CASE m_stepRun OF
	0:;
	5:  init(m_armNum);
		m_stepRun:=10;
	10: m_initFinishPID[m_armNum]:=armMotorRun();
	    IF m_step=0 THEN
			IF m_motorErrNum<>0 THEN
				m_errNum:=m_motorErrNum+m_armNum*1000;
			END_IF
			m_stepRun:=15;
		END_IF
	15: m_stepRun:=5;
		m_armNum:=m_armNum+1;
		IF m_armNum>=g_sArmNum THEN
			m_stepRun:=20;
		END_IF
	20: 
		FOR i:=1 TO g_sArmNum DO
			IF NOT m_initFinishPID[i] THEN
				m_isFinished:=10;
			END_IF
		END_FOR
		m_stepRun:=25;
	25:
		IF m_isFinished=5 THEN
			robotMotorRun:=TRUE;
			m_robotMotorRunMid:=TRUE;
		ELSE
			robotMotorRun:=FALSE;
			m_robotMotorRunMid:=TRUE;
		END_IF
		m_stepRun:=0;
END_CASE
robotMotorRun:=m_robotMotorRunMid;
END_METHOD

END_FUNCTION_BLOCK

// ---- FBs_Auxiliary/FB_Timer.TcPOU
FUNCTION_BLOCK FB_Timer
VAR
	fb_tonTimer:TON;
	tTime: TIME;
	tTimeMid: TIME;
	uiTime:UINT;
END_VAR

METHOD init : BOOL
tTimeMid:=T#0S;
fb_tonTimer(IN :=0);
END_METHOD

METHOD timer : BOOL
VAR_INPUT
	bStart: BOOL;
END_VAR
VAR_OUTPUT
	uiTimeHour: UINT;
	uiTimeMinute: UINT;
	uiTimeSecond: UINT;
END_VAR
fb_tonTimer(IN:=bStart, PT:=T#999H , );
IF NOT fb_tonTimer.IN THEN
	tTimeMid:=tTime;
END_IF	

tTime:=fb_tonTimer.ET+tTimeMid;
uiTime:=DT_TO_UINT(TIME_TO_DT(tTime));
uiTimeHour:= uiTime/3600;
uiTimeMinute:= uiTime/60-uiTimeHour*60;
uiTimeSecond:= uiTime-uiTimeHour*3600-uiTimeMinute*60;
END_METHOD

END_FUNCTION_BLOCK

// ---- FBs_Auxiliary/FB_PanelDetect.TcPOU
FUNCTION_BLOCK FB_PanelDetect
VAR_INPUT
END_VAR
VAR_OUTPUT
END_VAR
VAR
	m_panelOnCounts :INT :=0;
	m_panelOnCountThres :INT :=50;
END_VAR

// check if panel is on
METHOD run : BOOL
VAR_INPUT
	IOValue :UDINT;
END_VAR
//Panel single  At installation--2#0000   not installation --2#0101
IF (IOValue AND 16#06) = 6 THEN
	m_panelOnCounts := MIN( m_panelOnCounts +1,m_panelOnCountThres);
ELSIF (IOValue AND 16#06) = 0  THEN
	m_panelOnCounts :=0;
END_IF
run := m_panelOnCounts >= m_panelOnCountThres;
END_METHOD

END_FUNCTION_BLOCK

// ---- FBs_Auxiliary/FB_InstrumentDetect.TcPOU
FUNCTION_BLOCK FB_InstrumentDetect
VAR_INPUT
END_VAR
VAR_OUTPUT
END_VAR
VAR
	m_instruOnCounts :INT :=0;
	m_InstruOnCountThres :INT :=50;
END_VAR

// check if instrument is on
METHOD run : BOOL
VAR_INPUT
	IOValue :UDINT;
END_VAR
//Instrument single   At installation--2#0*0*   not installation --2#1*1*  And Hall single --2#100 0000
IF (IOValue AND 10#9) = 9  THEN
	m_instruOnCounts := MIN( m_instruOnCounts +1,m_InstruOnCountThres);
ELSIF (IOValue AND 10#9) = 0  THEN
	m_instruOnCounts :=0;
END_IF
run := m_instruOnCounts >= m_InstruOnCountThres;
END_METHOD

END_FUNCTION_BLOCK

// ---- FBs_BasicControllers/FB_BasicInstruControl.TcPOU
// instrument joints control
FUNCTION_BLOCK FB_BasicInstruControl
VAR_INPUT
END_VAR
VAR_OUTPUT
END_VAR
VAR
	// instrument PID control paramters
	m_instruKp:ARRAY[1..5] OF LREAL:=[5(2)];
	m_instruKd:ARRAY[1..5] OF LREAL:=[5(0.04)];
	m_instruKi:ARRAY[1..5] OF LREAL:=[5(5.0)];
	m_instruKiLimit:ARRAY[1..5] OF LREAL:=[5(250.0)];
	m_instruCtrlLimit:ARRAY[1..5] OF LREAL:=[5(540.0)];
	
	
	// gripper force level threshold for variable PID parameter
	m_forceLevelThres : ARRAY[1..3] OF LREAL := [40, 70, 101];
	
	// yaw PID control (when fingers grasp with force)
	m_yawKp:ARRAY[1..3] OF LREAL:=[2, 2, 2];
	m_yawKd:ARRAY[1..3] OF LREAL:=[0.04, 0.04, 0.04];
	m_yawKi:ARRAY[1..3] OF LREAL:=[2, 4, 6];
	m_yawKiLimit:LREAL:=250.0;
	m_yawCtrlLimit:LREAL:=540.0;
	
	// max grip force/current(mA)
	m_maxGripForce:LREAL;
	m_maxGripCurrent:LREAL:=450.0;
	
	// max gripper finger control force/current(mA)
	m_maxGripCtrlForce:LREAL;
	m_maxGripCtrlCurrent:LREAL:=650.0;
	
	// PID for instrument joint position
	m_instruJntCtrl:ARRAY[1..5] OF FB_PID;

	// PID for instrument yaw angle 
	m_instruYawCtrl : FB_PID;
	
	// command instrument joint position and velocity
	m_instruCmdJntPos:Vec5d;
	m_instruCmdJntVel:Vec5d;
	
	// current instrument joint position and velocity
	m_instruCurJntPos: Vec5d;
	m_instruCurJntVel:Vec5d;
	
	// grasp force level
	m_graspForceLevel:Lreal :=0;
	
	// ratio convert motor current to joint troque
	m_currentRatioMotor2Jnt:LREAL;
	
	// instrument joint control torque(when gripper is open)
	m_instruJntCtrlTrq:Vec5d:=[5(0.0)];

	// instrument yaw control torque(when gripper is closed)
	m_instruYawCtrlTrq:LREAL;
		
	// current gripper yaw velocity
	m_instruCurYawVel:LREAL;
	
	// yaw angle error(deg)
	m_yawAngErr : LREAL;
	
	// backlash compensation variables
	m_jntBacklash:ARRAY[1..5] OF LREAL:=[5(0)];
	m_instruLastCmdJntPos:Vec5d;
	
	// grip yaw compensation variables
 	m_gripYawCompAng :LREAL;
 	m_maxGripYawCompAng :LREAL;
	m_lastCmdYawAng:LREAL;
	m_jntMoveStep:LREAL := 0.5*g_deg2Rad;
	
END_VAR

METHOD calcBacklash : BOOL
VAR_IN_OUT CONSTANT
	// instrument joint command position
	i_cmdInstruJntPos :Vec5d;
	
	// command yaw position
	i_cmdYawPos : LREAL;
	
	// slave arm data
	i_slaveArm :FB_SlaveArm;
END_VAR

VAR
	i:INT;
	deltaAng:LREAL;
	maxBacklash: LREAL;
END_VAR
// backslash compensation
FOR i:=1 TO 4 DO
	// integral compensated backslash angle
	deltaAng:=i_cmdInstruJntPos[i]-m_instruLastCmdJntPos[i];
	IF ABS(deltaAng)>m_jntMoveStep THEN
		IF InstruType_PottsScissors = i_slaveArm.instrument.instruTypeInfo.m_InstruID THEN
			m_jntBacklash [i] := sign(deltaAng) * i_slaveArm.instrument.instruTypeInfo.m_instruYawBacklash;
		ELSE
			m_jntBacklash [i] := m_jntBacklash [i] + m_jntMoveStep*sign(deltaAng);
		END_IF
		m_instruLastCmdJntPos[i] := i_cmdInstruJntPos[i];
	END_IF
END_FOR


// exert grip force 
IF m_graspForceLevel >0  THEN
	
	// clear grip finger backlash
	m_jntBacklash [1]:=0;
	m_jntBacklash [2]:=0;
	
	// determin max compensated angle based on grip force 
	FOR i:=1 TO 4 DO 
		IF m_graspForceLevel<= g_instruGripYawCompForceLevel[i] THEN
			m_maxGripYawCompAng := g_instruGripYawCompAng[i];
			EXIT;
		END_IF
	END_FOR

	// compensate yaw joint angle in case it's driven by force difference between two fingers
	IF m_graspForceLevel > 80 AND  ABS(i_cmdYawPos - m_lastCmdYawAng) > m_jntMoveStep  THEN
		m_jntBacklash [3] := m_jntBacklash [3] -  4*m_jntMoveStep*sign(i_cmdYawPos - m_lastCmdYawAng);
	END_IF
	
	// determin  compensated angle
	IF ABS(i_cmdYawPos - m_lastCmdYawAng) > m_jntMoveStep  THEN
		// determin  compensated yaw  angle
		IF (i_cmdYawPos - m_lastCmdYawAng) * m_gripYawCompAng <= 0 THEN
			m_gripYawCompAng := m_gripYawCompAng + 4*m_jntMoveStep * sign(i_cmdYawPos-m_lastCmdYawAng);
		ELSE
			m_gripYawCompAng := m_gripYawCompAng + 2*m_jntMoveStep * sign(i_cmdYawPos-m_lastCmdYawAng);
		END_IF
		m_lastCmdYawAng := i_cmdYawPos;
	END_IF
	m_gripYawCompAng := LIMIT(-m_maxGripYawCompAng, m_gripYawCompAng,m_maxGripYawCompAng);
	

ELSE
	m_gripYawCompAng:=0;
	m_lastCmdYawAng := i_cmdYawPos;
END_IF

// limit compensated backslash angle
FOR i:=1 TO 4 DO
	IF i<3 THEN 
		maxBacklash:=i_slaveArm.instrument.instruTypeInfo.m_instruYawBacklash;
	ELSIF i=3 THEN
		maxBacklash:=i_slaveArm.instrument.instruTypeInfo.m_instruPitchBachlash;
	ELSIF i=4 THEN
		maxBacklash:=5.0*g_deg2Rad;
	ELSE
		maxBacklash:=0;
	END_IF
	
	IF GVL_InstruTestUIVars.g_enableRDCompensation THEN 
		GVL_InstruTestUIVars.g_enableBackendCompensation:=0;
		IF InstruType_ProGraspForceps = i_slaveArm.instrument.onChipData.m_InstruID THEN
			IF i<3 THEN 
				maxBacklash:=ASIN((2.8/5.26) * SIN(GVL_InstruTestUIVars.g_compensationAngleDH[2]*i_slaveArm.instrument.instruTypeInfo.m_k2*g_deg2Rad));
			ELSIF i=3 THEN
				maxBacklash:=ASIN((2.8/5.26) * SIN(GVL_InstruTestUIVars.g_compensationAngleDH[1]*i_slaveArm.instrument.instruTypeInfo.m_k1*g_deg2Rad));
			ELSIF i=4 THEN
				maxBacklash:=ASIN((2.8/5.26) * SIN(GVL_InstruTestUIVars.g_compensationAngleDH[3]*i_slaveArm.instrument.instruTypeInfo.m_k3*g_deg2Rad));
			ELSE
				maxBacklash:=0;
			END_IF
		ELSE
			IF i<3 THEN 
				maxBacklash:=GVL_InstruTestUIVars.g_compensationAngleDH[2]*g_deg2Rad*i_slaveArm.instrument.instruTypeInfo.m_k2;
			ELSIF i=3 THEN
				maxBacklash:=GVL_InstruTestUIVars.g_compensationAngleDH[1]*g_deg2Rad*i_slaveArm.instrument.instruTypeInfo.m_k1;
			ELSIF i=4 THEN
				maxBacklash:=GVL_InstruTestUIVars.g_compensationAngleDH[3]*g_deg2Rad*i_slaveArm.instrument.instruTypeInfo.m_k3;
			ELSE
				maxBacklash:=0;
			END_IF
		END_IF
	END_IF
	
	IF g_instruBacklashDir[i] > 0 THEN
		m_jntBacklash [i] := LIMIT(0, m_jntBacklash[i], maxBacklash);
	ELSE
		m_jntBacklash [i] := LIMIT(-maxBacklash, m_jntBacklash[i], 0);	
	END_IF
	
	IF GVL_InstruTestUIVars.g_enableBackendCompensation THEN 
		m_jntBacklash [i] := 0;
	END_IF
	
END_FOR
END_METHOD

METHOD init : BOOL
VAR_IN_OUT CONSTANT
	i_slaveArm:FB_SlaveArm;
	i_maxGripCurrent : LREAL;
	i_maxGripCtrlCurrent : LREAL;
END_VAR

VAR
	i,j:INT;
END_VAR
m_graspForceLevel:=0;
//m_maxGripCurrent := i_maxGripCurrent;
//m_maxGripCtrlCurrent :=i_maxGripCtrlCurrent;
//m_yawKiLimit := i_maxGripCurrent;
//m_yawCtrlLimit := i_maxGripCtrlCurrent;
// init controller
m_maxGripCurrent:= i_slaveArm.instrument.instruTypeInfo.m_normGripTrq; 
m_currentRatioMotor2Jnt:=GVL_SlaveMotorParameters.g_motorTrqConst[4]*GVL_SlaveMotorParameters.g_motorReduction[4]/1000;
m_maxGripForce := m_maxGripCurrent * m_currentRatioMotor2Jnt;
m_maxGripCtrlForce := m_maxGripCtrlCurrent * m_currentRatioMotor2Jnt;
FOR i:=1 TO 4 DO
	m_jntBacklash[i] := 0;
	m_instruKiLimit[i] := i_maxGripCurrent;
	m_instruCtrlLimit[i] := i_maxGripCtrlCurrent;
	m_instruCmdJntPos[i]:=i_slaveArm.curJntPos[i+3];
	
	m_instruCmdJntVel[i]:=0;
	
	m_instruJntCtrl[i].init(g_slaveArmCtrlCycleTime,m_instruKp[i],m_instruKd[i],m_instruKi[i],
		m_instruKiLimit[i]* m_currentRatioMotor2Jnt,	m_instruCtrlLimit[i]*m_currentRatioMotor2Jnt);
	
	m_instruLastCmdJntPos[i]:=m_instruCmdJntPos[i];
END_FOR
m_instruYawCtrl.init(g_slaveArmCtrlCycleTime,m_yawKp[1],m_yawKd[1],m_yawKi[1],m_yawKiLimit*m_currentRatioMotor2Jnt, m_yawCtrlLimit*m_currentRatioMotor2Jnt);
END_METHOD

METHOD run : BOOL
VAR_IN_OUT CONSTANT
	// instrument joint command position
	i_cmdInstruJntPos :Vec5d;
	
	// instrument joint command velocity
	i_cmdInstruJntVel :Vec5d;
	
	// command yaw position
	i_cmdYawPos : LREAL;
	
	// command yaw velocity
	i_cmdYawVel :LREAL;
	
	// command grip force level
	i_cmdGripForceLevel:LREAL;
	
	// slave arm data
	i_slaveArm :FB_SlaveArm;
END_VAR

VAR_OUTPUT
	// joint control torque
	o_cmdJntTrq:Vec5d;
END_VAR

VAR
	i: INT;
	deltaAng:LREAL;
END_VAR
IF i_cmdGripForceLevel >0 THEN
	m_graspForceLevel:=LIMIT(0,i_cmdGripForceLevel ,  100)	;
ELSE
	m_graspForceLevel:=LIMIT(-100,i_cmdGripForceLevel ,  0)	;
END_IF

// calculate instrument backlash
calcBacklash(i_cmdInstruJntPos, i_cmdYawPos, i_slaveArm);

IF InstruType_ForceBipolar = i_slaveArm.instrument.instruTypeInfo.m_InstruID THEN
	IF GVL_InstruTestUIVars.g_forceBipolarMode THEN
		// calculate instrument backlash
		setMaxGripTrq(220.0 * 2.5);
	ELSE
		setMaxGripTrq(220.0);
	END_IF
ELSE
	setMaxGripTrq(450.0);
END_IF


// joint position control
FOR i:=1 TO 4 DO	
	m_instruCmdJntPos[i]:=i_cmdInstruJntPos[i];
	m_instruCmdJntVel[i]:=i_cmdInstruJntVel[i];
	m_instruCurJntPos[i]:=i_slaveArm.curJntPos[i+3];
	m_instruCurJntVel[i]:= i_slaveArm.curJntVel[i+3];
	m_instruJntCtrlTrq[i]:=m_instruJntCtrl[i].run(m_instruCmdJntPos[i] + m_jntBacklash[i] ,m_instruCurJntPos[i], m_instruCmdJntVel[i], m_instruCurJntVel[i]);
END_FOR
m_instruJntCtrlTrq[5]:=0;

m_instruCurYawVel :=i_slaveArm.curDHJntVel[6];
m_yawAngErr:=g_rad2Deg*(i_cmdYawPos-i_slaveArm.curDHJntPos[6]);


// exert grip force 
IF m_graspForceLevel >0  THEN
	
	// varialbe PID control based on different gripper force level
	FOR i:=1 TO 3 DO 
		IF m_graspForceLevel < m_forceLevelThres[i] THEN
			m_instruYawCtrl.setPIDParam(m_yawKp[i],m_yawKd[i],m_yawKi[i]);
			EXIT;
		END_IF
	END_FOR

	// yaw control
	m_instruYawCtrlTrq:=m_instruYawCtrl.run(i_cmdYawPos+m_gripYawCompAng,i_slaveArm.curDHJntPos[6],i_cmdYawVel, m_instruCurYawVel);

	// add feed forward grasp force
	m_instruJntCtrlTrq[1]:= m_maxGripForce*m_graspForceLevel/100.0 + m_instruYawCtrlTrq;
	m_instruJntCtrlTrq[2]:= m_maxGripForce*m_graspForceLevel/100.0 - m_instruYawCtrlTrq;
	m_instruJntCtrlTrq[1]:=LIMIT(-m_maxGripForce/10.0,m_instruJntCtrlTrq[1], m_maxGripCtrlForce);
	m_instruJntCtrlTrq[2]:=LIMIT(-m_maxGripForce/10.0,m_instruJntCtrlTrq[2], m_maxGripCtrlForce);
// JUST FOR TEST
ELSIF m_graspForceLevel <0 THEN 
	m_instruJntCtrlTrq[1]:= m_maxGripForce*m_graspForceLevel/100.0;
	m_instruJntCtrlTrq[2]:= m_maxGripForce*m_graspForceLevel/100.0;
END_IF

o_cmdJntTrq := m_instruJntCtrlTrq;
END_METHOD

METHOD setMaxGripTrq : BOOL
VAR_INPUT
	i_maxGripTrq:LREAL;
END_VAR
m_maxGripCurrent := i_maxGripTrq;
m_maxGripForce := m_maxGripCurrent * m_currentRatioMotor2Jnt;
END_METHOD

END_FUNCTION_BLOCK

// ---- FBs_Robots/FB_SlaveArm.TcPOU
FUNCTION_BLOCK FB_SlaveArm
VAR
	//
	M_TESTfLAG:BOOL:=FALSE;
	m_jnt5Planner:Cubic_Polynomial_Interpolation;
	m_initAngle,m_initVel,m_initAcc,m_initT:REAL;
	m_targetAngle,m_targetVel,m_targetAcc:REAL;
	m_cmdAngle,m_cmdVel,m_cmdAcc:REAL;
	m_initFlag:BOOL:=FALSE;
	m_finishFlag:BOOL:=TRUE;
	m_endT:REAL:=5;
	m_dT:REAL:=0.0025;
	m_T:REAL:=0;
	// arm index, from 1 to 4
	m_armIdx: INT;
	
	// joints
	m_joints :ARRAY[1..g_sJntNum] OF FB_SlaveJoint;
	
	//  panel and insturment detect
	m_panelInstrumentOnIO AT%I*	:UDINT;
	m_panelDetect :FB_PanelDetect;
	m_instruDetect :FB_InstrumentDetect;
	m_instruNearDetect :FB_InstruNearDetect;
	m_panelOnFlag :BOOL:=FALSE;
	m_instruOnFlag :BOOL:=FALSE;
	m_instruNearFlag :BOOL:=FALSE;

	
	// trocar and  adjust detect
	m_adjustIO AT%I* :UDINT;
	m_adjustDetect :FB_AdjustDetect;
	m_trocarDetect : FB_TrocarDetect;
	m_adjustOnFlag :BOOL;
	m_trocarOnFlag :BOOL :=FALSE;
	m_adjustFallEdge :BOOL:=false;
	m_adjustFallEdgeDetect : F_TRIG;
	
	//arm light out to drive
	m_lightIO AT %Q* :DINT;
	
	//endoscope type and posture switch
	m_endoscopeTypeSwitch : FB_IOToggleCheck;
	m_endoscopePostureSwitch : FB_IOToggleCheck;
	
	// instrument instance
	m_instrument : FB_Instrument;
	
	// instrument invasion depth before it's unmounted
	m_instruInvasionDepth :LREAL;

	// arm cartesian data, defined in each arm origin
	m_curCartPose	:ST_Frame;
	m_curCartTwist: Vec6d;
	m_cmdCartTwist :Vec6d;
	m_cmdCartPose:ST_Frame;
	
	// arm joint data
	m_curMotorPos :Vec8d;
	m_curLinkPos :Vec8d;
	m_curLinkSingle :Vec8d;
	m_curJntPos :Vec8d;
	m_curDHJntPos :Vec6d;
	m_curGripAngle :LREAL;
	m_curJntVel :Vec8d;
	m_curDHJntVel :Vec6d;
	m_curJntTrq :Vec8d;
	m_rawJntCurrent :Vec8d;
	m_filtJntCurrent :Vec8d;
	m_cmdJntTrq :Vec8d;
	m_cmdJntCurrent : Vec8d;
	m_cmdJntPos :Vec8d;
	m_cmdJntVel :Vec8d;
		
	// arm dynamic data
	m_jntGravity : Vec8d:=g_zeroVec8d;
	m_jntMassMat : Mat3d;
	
	// arm jacobian and inverse
	m_jaco : Mat6d;
	
	// simulated status
	m_simJntPos :Vec8d;
	m_simDHJntPos :Vec6d;
	m_simGripAngle :LREAL;
	m_simCartPose : ST_Frame;
	m_simJaco : Mat6d;
	m_simJacoInv :Mat6d;
	m_isSingularity:BOOL:=false;
	
	// joint position controller
	m_jntPIDCtrl :ARRAY[1..g_sJntNum] OF FB_PID;
	
	// rising edge generator for instrument information reading
	m_ReadLDP:R_TRIG;
	
	// code execute time measure
	m_codeTime : Profiler;

	// output arm light
	m_SdoWrite:ARRAY [1..2] OF FB_EcCoESdoWrite;
	
	//IP of operating arm
	m_armNetId:T_AmsNetId; 	
	
	//Joint port number
	m_jointAddrJ8:UINT;	
	m_jointAddrPbox:UINT;	
	m_autoLogoutTon: TON;
	g_autoLogOutTRIG: R_TRIG;
	m_logStep: INT;
	m_actualNum: INT;
	m_registerNum: INT;
	m_register: INT;
	m_accountRepeat:BOOL;
	g_targetRatedCurrent: ARRAY[1..g_sJntNum] OF LREAL := [8(800)];

	
	fbSocketConnect      :FB_SocketConnect;
	fbSocketSend         :FB_SocketSend;;;
	fbSocketReceive      :FB_SocketReceive;
	bExecute:BOOL := TRUE;
	hSocket:T_hSocket;
	arrSendData: ARRAY [0..240] OF BYTE ;
	arrReadData: ARRAY [0..240] OF BYTE ;//read
	arrRFIDData: ARRAY [0..240] OF BYTE ;
	bSend   :BOOL;
	bReceive:BOOL;
	iStepRFID: INT;
	uiRFIDReadSN: ULINT;
	iStepRFIDOnLine: INT;
	fbTonRFID: TON;
	fbTonRFIDOnLine: TON;
	fbTonRFIDOnLineStep: TON;	
	g_offLineRFID:BOOL;
	m_offLineRFID:BOOL;
	
	fbTonCLK1:TON;
	fbTonCLK2:TON;
	
	uiRFIDRead:ULINT;
	wCRCReadSum:ULINT;
	g_readedRFID:BOOL;
	fbTonReadData:TON;
	
	
	wCRC16:WORD;
	g_moveMode:INT;
	g_energyType:INT;
	uiRFIDWrite:UINT;
	g_writedRFID:BOOL;
	
	g_RFIDinstruSN:ULINT;
	
	SNMid:INT;
	g_informationVerificationPassed:BOOL;
	g_instruSN:ULINT;
	m_writeRFIDTimes:DINT;
	m_writeInstrument_pos_L1:LREAL;
	m_writeInstrument_pos_L2:LREAL;
	m_writeInstrument_pos_L3:LREAL;
	m_readRFIDTimes:DINT;
	m_readInstrument_pos_L1:LREAL;
	m_readInstrument_pos_L2:LREAL;
	m_readInstrument_pos_L3:LREAL;
	
	fbTonRFIDReaded:TON;
	stateMachineMid: E_SlaveArmState;

	g_lastInstruJntPos: Vec5d;
	fbTon: TON;
	fbTon_Logout: TON;
	startFlag:BOOL;
	m_writeSdoStart: BOOL;
	m_writeSdoTimeStart: BOOL;
	m_writeSdoFinished: BOOL;
	m_SNWritten: BOOL;
	m_SNWriteStart: BOOL;
	m_bReadRecipeStep:   INT := 1;
	m_saveAccount:BOOL;
	m_saveCaliLinkEncoder:BOOL;
	RecipeManCommands:   RecipeManCommands;
	m_writePurposeSdoStart: BOOL;
	m_getSysTime:GETSYSTEMTIME;
	m_fileTime:T_FILETIME;
	m_time:STRING;
	m_timeNow:TIMESTRUCT;
	//mes
	m_serialNumOld:STRING;
	m_curTestCyclesOld:INT;
END_VAR

PROPERTY adjustFallEdge : BOOL
GET
adjustFallEdge := m_adjustFallEdge;
END_GET
END_PROPERTY

PROPERTY adjustOn : bool
GET
adjustOn := m_adjustOnFlag;
END_GET
END_PROPERTY

PROPERTY armIdx : int
GET
armIdx:=m_armIdx;
END_GET
END_PROPERTY

METHOD PROTECTED calcJaco : BOOL
VAR_IN_OUT CONSTANT
	i_DHJntPos :Vec6d;
END_VAR
VAR_IN_OUT
	r_jaco :Mat6d;
END_VAR
VAR_INPUT
END_VAR

VAR
	d1, L, a, b :LREAL;
	q3:LREAL;

	c1,c2,c4,c5,c6,c7 :LREAL;
	s1,s2,s4,s5,s6,s7 :LREAL;

END_VAR
d1:=GVL_SlaveArmKinematic.g_d1;
L:=m_instrument.instruTypeInfo.m_rodLength;
a:=m_instrument.instruTypeInfo.m_headLength;
b:=m_instrument.instruTypeInfo.m_fingerLength;

q3:=i_DHJntPos[3];
c1:=COS(i_DHJntPos[1]);
c2:=COS(i_DHJntPos[2]);
c4:=COS(i_DHJntPos[4]);
c5:=COS(i_DHJntPos[5]);
c6:=COS(i_DHJntPos[6]);

s1:=SIN(i_DHJntPos[1]);
s2:=SIN(i_DHJntPos[2]);
s4:=SIN(i_DHJntPos[4]);
s5:=SIN(i_DHJntPos[5]);
s6:=SIN(i_DHJntPos[6]);

// jacobian with DH joints
r_jaco[1,1]:=b*(c6*(c5*(c1*s4 - c2*c4*s1) + s1*s2*s5) - s6*(c1*c4 + c2*s1*s4)) + a*(c5*(c1*s4 - c2*c4*s1) + s1*s2*s5) - L*s1*s2 + q3*s1*s2;
r_jaco[1,2]:=-c1*(a*(c2*s5 + c4*c5*s2) - L*c2 + q3*c2 + b*(c6*(c2*s5 + c4*c5*s2) + s2*s4*s6));
r_jaco[1,3]:=-c1*s2;
r_jaco[1,4]:=s1*s2*(a*(c2*s5 + c4*c5*s2) + b*(c6*(c2*s5 + c4*c5*s2) + s2*s4*s6)) - c2*(b*(c6*(c5*(c1*s4 - c2*c4*s1) + s1*s2*s5) - s6*(c1*c4 + c2*s1*s4)) + a*(c5*(c1*s4 - c2*c4*s1) + s1*s2*s5));
r_jaco[1,5]:=- (a*(c2*s5 + c4*c5*s2) + b*(c6*(c2*s5 + c4*c5*s2) + s2*s4*s6))*(c1*c4 + c2*s1*s4) - s2*s4*(b*(c6*(c5*(c1*s4 - c2*c4*s1) + s1*s2*s5) - s6*(c1*c4 + c2*s1*s4)) + a*(c5*(c1*s4 - c2*c4*s1) + s1*s2*s5));
r_jaco[1,6]:= b*(c6*(c5*(c1*s4 - c2*c4*s1) + s1*s2*s5) - s6*(c1*c4 + c2*s1*s4))*(c2*c5 - c4*s2*s5) + b*(s5*(c1*s4 - c2*c4*s1) - c5*s1*s2)*(c6*(c2*s5 + c4*c5*s2) + s2*s4*s6);


r_jaco[2,1]:=0;
r_jaco[2,2]:=c1*(a*(c5*(s1*s4 + c1*c2*c4) - c1*s2*s5) + b*(c6*(c5*(s1*s4 + c1*c2*c4) - c1*s2*s5) - s6*(c4*s1 - c1*c2*s4)) + L*c1*s2 - q3*c1*s2) - s1*(b*(c6*(c5*(c1*s4 - c2*c4*s1) + s1*s2*s5) - s6*(c1*c4 + c2*s1*s4)) + a*(c5*(c1*s4 - c2*c4*s1) + s1*s2*s5) - L*s1*s2 + q3*s1*s2);
r_jaco[2,3]:= c2;
r_jaco[2,4]:=- s1*s2*(a*(c5*(s1*s4 + c1*c2*c4) - c1*s2*s5) + b*(c6*(c5*(s1*s4 + c1*c2*c4) - c1*s2*s5) - s6*(c4*s1 - c1*c2*s4))) - c1*s2*(b*(c6*(c5*(c1*s4 - c2*c4*s1) + s1*s2*s5) - s6*(c1*c4 + c2*s1*s4)) + a*(c5*(c1*s4 - c2*c4*s1) + s1*s2*s5));
r_jaco[2,5]:=(a*(c5*(s1*s4 + c1*c2*c4) - c1*s2*s5) + b*(c6*(c5*(s1*s4 + c1*c2*c4) - c1*s2*s5) - s6*(c4*s1 - c1*c2*s4)))*(c1*c4 + c2*s1*s4) - (b*(c6*(c5*(c1*s4 - c2*c4*s1) + s1*s2*s5) - s6*(c1*c4 + c2*s1*s4)) + a*(c5*(c1*s4 - c2*c4*s1) + s1*s2*s5))*(c4*s1 - c1*c2*s4);
r_jaco[2,6]:=b*(c6*(c5*(c1*s4 - c2*c4*s1) + s1*s2*s5) - s6*(c1*c4 + c2*s1*s4))*(s5*(s1*s4 + c1*c2*c4) + c1*c5*s2) - b*(s5*(c1*s4 - c2*c4*s1) - c5*s1*s2)*(c6*(c5*(s1*s4 + c1*c2*c4) - c1*s2*s5) - s6*(c4*s1 - c1*c2*s4));

r_jaco[3,1]:=a*(c5*(s1*s4 + c1*c2*c4) - c1*s2*s5) + b*(c6*(c5*(s1*s4 + c1*c2*c4) - c1*s2*s5) - s6*(c4*s1 - c1*c2*s4)) + L*c1*s2 - q3*c1*s2;
r_jaco[3,2]:=-s1*(a*(c2*s5 + c4*c5*s2) - L*c2 + q3*c2 + b*(c6*(c2*s5 + c4*c5*s2) + s2*s4*s6));
r_jaco[3,3]:=-s1*s2;
r_jaco[3,4]:=- c2*(a*(c5*(s1*s4 + c1*c2*c4) - c1*s2*s5) + b*(c6*(c5*(s1*s4 + c1*c2*c4) - c1*s2*s5) - s6*(c4*s1 - c1*c2*s4))) - c1*s2*(a*(c2*s5 + c4*c5*s2) + b*(c6*(c2*s5 + c4*c5*s2) + s2*s4*s6));
r_jaco[3,5]:=- (a*(c2*s5 + c4*c5*s2) + b*(c6*(c2*s5 + c4*c5*s2) + s2*s4*s6))*(c4*s1 - c1*c2*s4) - s2*s4*(a*(c5*(s1*s4 + c1*c2*c4) - c1*s2*s5) + b*(c6*(c5*(s1*s4 + c1*c2*c4) - c1*s2*s5) - s6*(c4*s1 - c1*c2*s4)));
r_jaco[3,6]:=b*(c6*(c5*(s1*s4 + c1*c2*c4) - c1*s2*s5) - s6*(c4*s1 - c1*c2*s4))*(c2*c5 - c4*s2*s5) + b*(c6*(c2*s5 + c4*c5*s2) + s2*s4*s6)*(s5*(s1*s4 + c1*c2*c4) + c1*c5*s2);

r_jaco[4,1]:=0;
r_jaco[4,2]:=-s1;
r_jaco[4,3]:=0;
r_jaco[4,4]:=-c1*s2;
r_jaco[4,5]:=c1*c2*s4 - c4*s1;
r_jaco[4,6]:=s5*(s1*s4 + c1*c2*c4) + c1*c5*s2;

r_jaco[5,1]:=-1;
r_jaco[5,2]:=0;
r_jaco[5,3]:=0;
r_jaco[5,4]:=c2;
r_jaco[5,5]:=s2*s4;
r_jaco[5,6]:=c4*s2*s5 - c2*c5;

r_jaco[6,1]:=0;
r_jaco[6,2]:=c1;
r_jaco[6,3]:=0;
r_jaco[6,4]:=-s1*s2;
r_jaco[6,5]:=c1*c4 + c2*s1*s4;
r_jaco[6,6]:=c5*s1*s2 - s5*(c1*s4 - c2*c4*s1);
END_METHOD

METHOD PROTECTED checkIO : BOOL

VAR

	i: INT;
	ReturnDwordRead:DWORD;
	ReturnDwordWrite:DWORD;
END_VAR
// check adjust button
m_adjustOnFlag := m_adjustDetect.run(m_adjustIO);
m_adjustFallEdgeDetect(CLK:=m_adjustOnFlag, Q=>m_adjustFallEdge);

// check trocar
m_trocarOnFlag := m_trocarDetect.run(m_adjustIO);

// check panel and instrument
m_panelOnFlag := m_panelDetect.run(m_panelInstrumentOnIO);
m_instruOnFlag :=m_instruDetect.run(m_panelInstrumentOnIO);
m_instruNearFlag := m_instruNearDetect.run(m_panelInstrumentOnIO);

//read instrument information
IF FALSE = m_instruOnFlag THEN
	m_instrument.reset();
END_IF


m_ReadLDP(CLK:= m_instruOnFlag, Q=>startFlag );
// try to read again if instrument ID is undefined
startFlag := startFlag OR m_instrument.onChipData.m_ErrorID = 1 OR GVL_InstruTestUIVars.g_readInstruinformation;
m_instrument.readParameters(startFlag);

GVL_InstruTestUIVars.g_readInstruinformationFlag:=m_instrument.onChipData.m_InstruReadSucceed;
// check endoscope type and posture 
IF m_endoscopeTypeSwitch.check((m_panelInstrumentOnIO AND 16#20)=32) THEN
	IF m_instrument.curScopeType = EndoScopeType_30 THEN
		m_instrument.nextScopeType := EndoscopeType_0;
	ELSE
		m_instrument.nextScopeType := EndoscopeType_30;
	END_IF
END_IF
IF m_endoscopePostureSwitch.check((m_panelInstrumentOnIO AND 16#10)=16) AND m_instrument.curScopeType = EndoScopeType_30  THEN
	IF m_instrument.curScopePosture = EndoScopePosture_HeadDown THEN
		m_instrument.nextScopePosture := EndoscopePosture_HeadUp;
	ELSE
		m_instrument.nextScopePosture := EndoScopePosture_HeadDown;
	END_IF
END_IF

IF GVL_InstruTestUIVars.g_incInstruNumOfUses THEN
	GVL_InstruTestUIVars.g_jnt5RotateFlag:=TRUE;
	m_writeSdoTimeStart := TRUE;
ELSE
	IF m_writeSdoTimeStart THEN
		IF   NOT m_writeSdoFinished THEN
			m_writeSdoFinished :=instrument.addNumOfUseToChip();

		ELSE
			m_writeSdoTimeStart :=FALSE;
			m_writeSdoFinished:=FALSE;
		END_IF
	END_IF
END_IF

IF GVL_InstruTestUIVars.g_clearInstruNumOfUses THEN
	m_writeSdoStart := TRUE;
ELSE
	IF m_writeSdoStart THEN
		IF   NOT m_writeSdoFinished THEN
			m_writeSdoFinished :=instrument.clearNumOfUseToChip();

		ELSE
			m_writeSdoStart :=FALSE;
			m_writeSdoFinished:=FALSE;
		END_IF
	END_IF
END_IF

// write SN to CoE
IF GVL_InstruTestUIVars.g_writeSNFlag THEN
	m_SNWriteStart := TRUE;
ELSE
	IF m_SNWriteStart THEN
		IF   NOT m_SNWritten THEN
			m_SNWritten := instrument.writeSNToChip(STRING_TO_ULINT(GVL_InstruTestUIVars.g_newInstruSN));
		ELSE
			m_SNWriteStart :=FALSE;
			m_SNWritten:=FALSE;
		END_IF
	END_IF
END_IF

IF GVL_InstruTestUIVars.g_writeInstruPurpose AND m_instrument.onChipData.m_InstruReadSucceed THEN
	m_writePurposeSdoStart := TRUE;
ELSE
	IF m_writePurposeSdoStart THEN
		IF   NOT m_writeSdoFinished THEN
			m_writeSdoFinished :=instrument.writePurpose();

		ELSE
			m_writePurposeSdoStart :=FALSE;
			m_writeSdoFinished:=FALSE;
		END_IF
	END_IF
END_IF

GVL_InstruTestUIVars.g_maxAngle:=INT_TO_REAL(REAL_TO_INT(m_instrument.instruTypeInfo.m_maxGripAngle/g_deg2Rad));
GVL_InstruTestUIVars.g_maxRoll:=INT_TO_REAL(REAL_TO_INT(m_instrument.instruTypeInfo.m_rollLimit/g_deg2Rad));
GVL_InstruTestUIVars.g_maxPitch:=INT_TO_REAL(REAL_TO_INT(m_instrument.instruTypeInfo.m_pitchLimit/g_deg2Rad));
GVL_InstruTestUIVars.g_maxYaw:=INT_TO_REAL(REAL_TO_INT(m_instrument.instruTypeInfo.m_yawLimit/g_deg2Rad));
GVL_InstruTestUIVars.g_maxAngleEnable:=GVL_InstruTestUIVars.g_targetGripAng*g_deg2rad>m_instrument.instruTypeInfo.m_maxGripAngle;
GVL_InstruTestUIVars.g_maxRollEnable:=ABS(GVL_InstruTestUIVars.g_targetRollAng)*g_deg2rad>m_instrument.instruTypeInfo.m_rollLimit;
GVL_InstruTestUIVars.g_maxPitchEnable:=ABS(GVL_InstruTestUIVars.g_targetPitchAng)*g_deg2rad>m_instrument.instruTypeInfo.m_pitchLimit;
GVL_InstruTestUIVars.g_maxYawEnable:=ABS(GVL_InstruTestUIVars.g_targetYawAng)*g_deg2rad>m_instrument.instruTypeInfo.m_yawLimit;

GVL_InstruTestUIVars.g_incInstruNumOfUses:=FALSE;
GVL_InstruTestUIVars.g_clearInstruNumOfUses:=FALSE;
GVL_InstruTestUIVars.g_writeSNFlag:=FALSE;
GVL_InstruTestUIVars.g_writeInstruPurpose:=FALSE;

GVL_InstruTestUIVars.g_instruNumberOfUses:=ULINT_TO_UINT( m_instrument.onChipData.m_InstruusageCounts);
GVL_InstruTestUIVars.g_instruNumberOfAllUses:=ULINT_TO_UINT( m_instrument.onChipData.m_InstruUsageCounts);
GVL_InstruTestUIVars.g_readInstruPurpose:=ULINT_TO_UINT( m_instrument.onChipData.m_InstruPurpose);
GVL_InstruTestUIVars.g_readPurposeTime:=ULINT_TO_UINT( m_instrument.onChipData.m_InstruPurposeTime);

GVL_InstruTestUIVars.g_instruSN:=ULINT_TO_STRING(m_instrument.onChipData.m_InstruseriesNum);
IF (LEN(GVL_InstruTestUIVars.g_instruSN)=10)THEN
	GVL_InstruTestUIVars.g_instruSN:=concat('00',GVL_InstruTestUIVars.g_instruSN);
ELSIF  (LEN(GVL_InstruTestUIVars.g_instruSN)=11)THEN
	GVL_InstruTestUIVars.g_instruSN:=concat('0',GVL_InstruTestUIVars.g_instruSN);
ELSE
	GVL_InstruTestUIVars.g_instruSN:=GVL_InstruTestUIVars.g_instruSN;
END_IF

GVL_InstruTestUIVars.g_rotationActualCurrent:=m_filtJntCurrent[7];
GVL_InstruTestUIVars.g_pitchActualCurrent:=m_filtJntCurrent[6];
GVL_InstruTestUIVars.g_deviationActualCurrent:=m_filtJntCurrent[4];
//***************************修改电流极限**************************//
GVL_InstruTestUIVars.g_actualRatedCurrent:=g_targetRatedCurrent;
IF GVL_InstruTestUIVars.g_modifyRatedCurrent THEN
	GVL_InstruTestUIVars.g_modifyRatedCurrent:=FALSE;
	FOR i:=1 TO 8 BY 1 DO 
		GVL_InstruTestUIVars.g_actualRatedCurrent[i]:=GVL_InstruTestUIVars.g_targetRatedCurrent;
		g_targetRatedCurrent[i]:=GVL_InstruTestUIVars.g_targetRatedCurrent;
	END_FOR
END_IF
IF GVL_InstruTestUIVars.g_rotationTargetCurrent=0 THEN GVL_InstruTestUIVars.g_rotationTargetCurrent:=100; END_IF
IF GVL_InstruTestUIVars.g_pitchTargetCurrent=0 THEN GVL_InstruTestUIVars.g_pitchTargetCurrent:=100; END_IF
IF GVL_InstruTestUIVars.g_deviationTargetCurrent=0 THEN GVL_InstruTestUIVars.g_deviationTargetCurrent:=100; END_IF
IF GVL_InstruTestUIVars.g_deviationTargetCurrent=0 THEN GVL_InstruTestUIVars.g_deviationTargetCurrent:=100; END_IF
IF GVL_InstruTestUIVars.g_account.actualPermission=2 AND GVL_InstruTestUIVars.g_stateMachine=SlaveArmState_InstruManualTest  THEN
	GVL_InstruTestUIVars.g_actualRatedCurrent[7]:=GVL_InstruTestUIVars.g_rotationTargetCurrent;
	GVL_InstruTestUIVars.g_actualRatedCurrent[6]:=GVL_InstruTestUIVars.g_pitchTargetCurrent;
	GVL_InstruTestUIVars.g_actualRatedCurrent[5]:=GVL_InstruTestUIVars.g_deviationTargetCurrent;
	GVL_InstruTestUIVars.g_actualRatedCurrent[4]:=GVL_InstruTestUIVars.g_deviationTargetCurrent;
END_IF
IF GVL_InstruTestUIVars.g_stateMachine=SlaveArmState_InstruAutoTest AND GVL_MES.g_autoTestMode=3 THEN
	GVL_InstruTestUIVars.g_actualRatedCurrent[4]:=540;
	GVL_InstruTestUIVars.g_actualRatedCurrent[5]:=540;
	GVL_InstruTestUIVars.g_actualRatedCurrent[6]:=540;
	GVL_InstruTestUIVars.g_actualRatedCurrent[7]:=540;
	IF m_instrument.onChipData.m_InstruReadSucceed AND(InstruType_CauteryHook=m_instrument.m_instruType OR InstruType_CauterySpatula=m_instrument.m_instruType) THEN
	GVL_InstruTestUIVars.g_actualRatedCurrent[4]:=270;
	GVL_InstruTestUIVars.g_actualRatedCurrent[5]:=270;
	GVL_InstruTestUIVars.g_actualRatedCurrent[6]:=270;
	GVL_InstruTestUIVars.g_actualRatedCurrent[7]:=270;
	END_IF
END_IF
//Account
GVL_InstruTestUIVars.g_account.memoryAccountNumber[0] :='admin';
GVL_InstruTestUIVars.g_account.memoryPassWord[0] :='yfAGIBOT2025';
GVL_InstruTestUIVars.g_account.memoryPermission[0] :=1;
GVL_InstruTestUIVars.g_account.memoryName[0] :='admin';
GVL_InstruTestUIVars.g_account.memoryWorkNum[0] :=101;
GVL_InstruTestUIVars.g_account.memoryDisable[0]:=FALSE;
CASE m_logStep OF 
	0: 
	  IF GVL_InstruTestUIVars.g_account.logOn THEN 
		   m_logStep:=5;
		   m_actualNum:=-1;
		  GVL_InstruTestUIVars.g_account.logOn:=FALSE;
	  END_IF
	5:
	FOR i:= 0 TO 50 BY 1 DO
		IF GVL_InstruTestUIVars.g_account.actualAccountNumber = GVL_InstruTestUIVars.g_account.memoryAccountNumber[i] AND GVL_InstruTestUIVars.g_account.actualAccountNumber <> ''THEN
			m_actualNum:=i;
			m_logStep:=10;
		ELSE
			IF m_actualNum=-1 THEN
				GVL_InstruTestUIVars.g_account.prompt:='Account Err';
				m_logStep:=0;
			END_IF
		END_IF
	END_FOR
	10:
	IF GVL_InstruTestUIVars.g_account.actualPassWord = GVL_InstruTestUIVars.g_account.memoryPassWord[m_actualNum] AND GVL_InstruTestUIVars.g_account.actualAccountNumber <> ''THEN
		m_logStep:=12;
	ELSE
		GVL_InstruTestUIVars.g_account.prompt:='PassWord Err';
		m_logStep:=0;
	END_IF
	12:
	IF GVL_InstruTestUIVars.g_account.memoryDisable[m_actualNum] THEN
		GVL_InstruTestUIVars.g_account.prompt:='No Enable';
		m_logStep:=0;
	ELSE
		m_logStep:=15;
	END_IF
	15:
	GVL_InstruTestUIVars.g_account.actualPermission := GVL_InstruTestUIVars.g_account.memoryPermission[m_actualNum];
	GVL_InstruTestUIVars.g_account.actualWorkNum := GVL_InstruTestUIVars.g_account.memoryWorkNum[m_actualNum];
	GVL_InstruTestUIVars.g_account.actualName := GVL_InstruTestUIVars.g_account.memoryName[m_actualNum];
	GVL_InstruTestUIVars.g_account.autoLogOut:=FALSE;
	GVL_InstruTestUIVars.g_account.prompt:='Login Succeeded';
	m_logStep:=0;
END_CASE

FOR i:=1 TO 5 DO 
	IF stateMachineMid<>GVL_InstruTestUIVars.g_stateMachine OR ABS(GVL_InstruTestUIVars.g_curInstruJntPos[i]-g_lastInstruJntPos[i])>0.01 THEN
		GVL_InstruTestUIVars.g_account.autoLogOut:=FALSE;
	ELSE
		IF NOT GVL_InstruTestUIVars.g_account.autoLogOut THEN 
			IF fbTon_Logout.Q THEN
				GVL_InstruTestUIVars.g_account.autoLogOut:=TRUE;
			END_IF
		END_IF
	END_IF
END_FOR
	fbTon(IN:= NOT fbTon.Q, PT:=T#10MS );
	IF fbTon.Q THEN
		g_lastInstruJntPos:= GVL_InstruTestUIVars.g_curInstruJntPos;
	END_IF
stateMachineMid:=GVL_InstruTestUIVars.g_stateMachine;
fbTon_Logout(IN:=NOT GVL_InstruTestUIVars.g_account.autoLogOut,PT:=T#0.1S);


m_autoLogoutTon(IN:=GVL_InstruTestUIVars.g_account.autoLogOut,PT:=T#1H);
g_autoLogOutTRIG(CLK:=m_autoLogoutTon.Q);
IF GVL_InstruTestUIVars.g_account.logOut OR g_autoLogOutTRIG.Q THEN
	GVL_InstruTestUIVars.g_account.actualPermission :=0;
	GVL_InstruTestUIVars.g_account.actualAccountNumber :='';
	GVL_InstruTestUIVars.g_account.actualPassWord :='';
	GVL_InstruTestUIVars.g_account.actualWorkNum :=0;
	GVL_InstruTestUIVars.g_account.actualName :='';
	GVL_InstruTestUIVars.g_account.logOut:=FALSE;
	GVL_InstruTestUIVars.g_account.prompt:='';
END_IF
IF GVL_InstruTestUIVars.g_clearInformation THEN
	GVL_InstruTestUIVars.g_account.actualAccountNumber :='';
	GVL_InstruTestUIVars.g_account.actualPassWord :='';
	GVL_InstruTestUIVars.g_account.actualWorkNum :=0;
	GVL_InstruTestUIVars.g_account.actualName :='';
	GVL_InstruTestUIVars.g_account.prompt:='';
	GVL_InstruTestUIVars.g_account.registerAccountNumber :='';
	GVL_InstruTestUIVars.g_account.registerPassWord :='';
	GVL_InstruTestUIVars.g_account.registerWorkNum :=0;
	GVL_InstruTestUIVars.g_account.registerName :='';
	GVL_InstruTestUIVars.g_account.prompt:='';
	GVL_InstruTestUIVars.g_clearInformation:=FALSE;
END_IF
IF GVL_InstruTestUIVars.g_account.registerPermission<>2 AND GVL_InstruTestUIVars.g_account.registerPermission<>3 AND
	GVL_InstruTestUIVars.g_account.registerPermission<>4 THEN
//	GVL_InstruTestUIVars.g_account.registerPermission:=4;
END_IF
m_getSysTime(timeLoDW=>m_fileTime.dwLowDateTime, timeHiDW=>m_fileTime.dwHighDateTime);
m_timeNow:=FILETIME_TO_SYSTEMTIME(m_fileTime);
m_timeNow.wHour:=m_timeNow.wHour+8;
IF m_timeNow.wHour>23 THEN
	m_timeNow.wHour:=m_timeNow.wHour-24;
END_IF
m_time:=SYSTEMTIME_TO_STRING(m_timeNow);
CASE m_registerNum OF 
	0:
	  IF GVL_InstruTestUIVars.g_account.register THEN 
		  GVL_InstruTestUIVars.g_account.register:=FALSE;
		  GVL_InstruTestUIVars.g_account.prompt:='';
		  m_accountRepeat:=FALSE;
		  m_register:=-1;
		  m_registerNum:=5;
	  END_IF
	5:
	FOR i:= 0 TO 50 BY 1 DO
      IF  GVL_InstruTestUIVars.g_account.registerAccountNumber <> GVL_InstruTestUIVars.g_account.memoryAccountNumber[i] AND GVL_InstruTestUIVars.g_account.registerAccountNumber <> ''THEN
		;	  
	  ELSE
		  m_accountRepeat:=TRUE;
	  END_IF
	END_FOR
	m_registerNum:=6;
	6:
	IF m_accountRepeat THEN
		GVL_InstruTestUIVars.g_account.prompt:='Account Repeat';
		m_registerNum:=0;
	ELSE
		m_registerNum:=10;
	END_IF
	10:
	IF GVL_InstruTestUIVars.g_account.registerPassWord<> '' THEN
		m_registerNum:=15;
	ELSE
		GVL_InstruTestUIVars.g_account.prompt:='No PassWord';
		m_registerNum:=0;
	END_IF
	15:
	IF GVL_InstruTestUIVars.g_account.registerWorkNum<> 0 THEN
		m_registerNum:=20;
	ELSE
		GVL_InstruTestUIVars.g_account.prompt:='No WorkNum';
		m_registerNum:=0;
	END_IF
	20:
	IF GVL_InstruTestUIVars.g_account.registerName<> '' THEN
		m_registerNum:=25;
	ELSE
		GVL_InstruTestUIVars.g_account.prompt:='No Name';
		m_registerNum:=0;
	END_IF
	25:
	IF GVL_InstruTestUIVars.g_account.registerPermission<> 0 THEN
		m_registerNum:=30;
	ELSE
		GVL_InstruTestUIVars.g_account.prompt:='No Permission';
		m_registerNum:=0;
	END_IF
	30:
	FOR i:= 50 TO 0 BY -1 DO
      IF  '' = GVL_InstruTestUIVars.g_account.memoryAccountNumber[i] THEN
		 m_register:=i;
		 m_registerNum:=35;
	  ELSE
		  IF m_register=-1 THEN
			 GVL_InstruTestUIVars.g_account.prompt:='No Room';
			 m_registerNum:=0;	
		END_IF
	  END_IF
 	END_FOR
	35:
	GVL_InstruTestUIVars.g_account.memoryAccountNumber[m_register]:=GVL_InstruTestUIVars.g_account.registerAccountNumber;
	GVL_InstruTestUIVars.g_account.memoryPassWord[m_register]:=GVL_InstruTestUIVars.g_account.registerPassWord;
	GVL_InstruTestUIVars.g_account.memoryWorkNum[m_register]:=GVL_InstruTestUIVars.g_account.registerWorkNum;
	GVL_InstruTestUIVars.g_account.memoryName[m_register]:=GVL_InstruTestUIVars.g_account.registerName;
	GVL_InstruTestUIVars.g_account.memoryPermission[m_register]:=GVL_InstruTestUIVars.g_account.registerPermission;
	IF GVL_InstruTestUIVars.g_account.registerPermission=1 THEN
		GVL_InstruTestUIVars.g_account.memoryPermission[m_register]:=4;
	END_IF
	GVL_InstruTestUIVars.g_account.memoryTime[m_register]:=m_time;
	GVL_InstruTestUIVars.g_account.prompt:='Register Succeeded';
	m_registerNum:=0;
	m_saveAccount:=TRUE;
END_CASE

GVL_InstruTestUIVars.g_accountSN := LIMIT(1,GVL_InstruTestUIVars.g_accountSN, 50);
IF GVL_InstruTestUIVars.g_accountDelete THEN 
	GVL_InstruTestUIVars.g_accountDelete:=FALSE;
	m_saveAccount:=TRUE;
	GVL_InstruTestUIVars.g_account.memoryAccountNumber[GVL_InstruTestUIVars.g_accountSN]:='';
	GVL_InstruTestUIVars.g_account.memoryPassWord[GVL_InstruTestUIVars.g_accountSN]:='';
	GVL_InstruTestUIVars.g_account.memoryWorkNum[GVL_InstruTestUIVars.g_accountSN]:=0;
	GVL_InstruTestUIVars.g_account.memoryName[GVL_InstruTestUIVars.g_accountSN]:='';
	GVL_InstruTestUIVars.g_account.memoryPermission[GVL_InstruTestUIVars.g_accountSN]:=0;
	GVL_InstruTestUIVars.g_account.memoryTime[GVL_InstruTestUIVars.g_accountSN]:='';
END_IF
IF GVL_InstruTestUIVars.g_disableAccount THEN 
	GVL_InstruTestUIVars.g_disableAccount:=FALSE;
	IF GVL_InstruTestUIVars.g_account.memoryDisable[GVL_InstruTestUIVars.g_accountSN] THEN
		GVL_InstruTestUIVars.g_account.memoryDisable[GVL_InstruTestUIVars.g_accountSN]:=FALSE;
	ELSE
		GVL_InstruTestUIVars.g_account.memoryDisable[GVL_InstruTestUIVars.g_accountSN]:=TRUE;
	END_IF
END_IF	
FOR i:=1 TO 50 BY 1 DO 
	IF GVL_InstruTestUIVars.g_account.memoryAccountNumber[i]='' THEN
		GVL_InstruTestUIVars.g_account.memoryDisable[i]:=FALSE;
	END_IF
END_FOR
GVL_InstruTestUIVars.g_queryAccountSN := LIMIT(0,GVL_InstruTestUIVars.g_queryAccountSN, 50);
IF GVL_InstruTestUIVars.g_queryAccountFlag THEN 
	GVL_InstruTestUIVars.g_queryAccountFlag:=FALSE;
	GVL_InstruTestUIVars.g_queryAccountNumber:='';
	GVL_InstruTestUIVars.g_queryPassWord:='';
	GVL_InstruTestUIVars.g_queryPermission:=0;
	GVL_InstruTestUIVars.g_queryWorkNum:=0;
	GVL_InstruTestUIVars.g_queryName:='';
	GVL_InstruTestUIVars.g_queryTime:='';
	GVL_InstruTestUIVars.g_queryAccountNumber:=GVL_InstruTestUIVars.g_account.memoryAccountNumber[GVL_InstruTestUIVars.g_queryAccountSN];
	GVL_InstruTestUIVars.g_queryPassWord:=GVL_InstruTestUIVars.g_account.memoryPassWord[GVL_InstruTestUIVars.g_queryAccountSN];
	GVL_InstruTestUIVars.g_queryPermission:=GVL_InstruTestUIVars.g_account.memoryPermission[GVL_InstruTestUIVars.g_queryAccountSN];
	GVL_InstruTestUIVars.g_queryWorkNum:=GVL_InstruTestUIVars.g_account.memoryWorkNum[GVL_InstruTestUIVars.g_queryAccountSN];
	GVL_InstruTestUIVars.g_queryName:=GVL_InstruTestUIVars.g_account.memoryName[GVL_InstruTestUIVars.g_queryAccountSN];
	GVL_InstruTestUIVars.g_queryTime:=GVL_InstruTestUIVars.g_account.memoryTime[GVL_InstruTestUIVars.g_queryAccountSN];
END_IF
IF GVL_InstruTestUIVars.g_queryClear THEN 
	GVL_InstruTestUIVars.g_queryClear:=FALSE;
	GVL_InstruTestUIVars.g_queryAccountNumber:='';
	GVL_InstruTestUIVars.g_queryPassWord:='';
	GVL_InstruTestUIVars.g_queryPermission:=0;
	GVL_InstruTestUIVars.g_queryWorkNum:=0;
	GVL_InstruTestUIVars.g_queryName:='';
	GVL_InstruTestUIVars.g_queryTime:='';
END_IF

bExecute:=NOT fbSocketConnect.bError OR fbTon.Q;

fbSocketConnect(
	sSrvNetId:= , 
	sRemoteHost:='192.168.1.202' , 
	nRemotePort:= 4196, 
	bExecute:= bExecute, 
	tTimeout:=T#3S , 
	bBusy=> , 
	bError=> , 
	nErrId=> , 
	hSocket=>hSocket );
	
	fbSocketSend(
	sSrvNetId:= , 
	hSocket:= hSocket, 
	cbLen:= SIZEOF(arrSendData), 
	pSrc:= ADR(arrSendData), 
	bExecute:= bSend, 
	tTimeout:= T#3S, 
	bBusy=> , 
	bError=> , 
	nErrId=> );
	
	
	fbSocketReceive(
	sSrvNetId:= , 
	hSocket:=hSocket , 
	cbLen:= SIZEOF(arrReadData), 
	pDest:= ADR(arrReadData), 
	bExecute:= bReceive, 
	tTimeout:= T#3S, 
	bBusy=> , 
	bError=> , 
	nErrId=> , 
	nRecBytes=> );
	
	bSend:=FALSE;
	fbTonCLK1(IN:=NOT fbTonCLK2.Q,PT:=T#1S);
	fbTonCLK2(IN:=fbTonCLK1.Q,PT:=T#1S);
	bReceive:=fbTonCLK1.Q;
//RFID
m_instrument.readParametersRFID(GVL_InstruTestUIVars.g_readRFID);
GVL_InstruTestUIVars.g_readRFID:=FALSE;
g_informationVerificationPassed:=FALSE;
IF m_instrument.onChipData.m_InstruReadSucceedRFID AND m_instrument.onChipData.m_InstruseriesNumRFID=m_instrument.onChipData.m_InstruseriesNum  AND 
	ABS(m_instrument.onChipData.m_InstruPosRFID[1]-m_instrument.onChipData.m_InstruPos[1])<0.01 AND
	ABS(m_instrument.onChipData.m_InstruPosRFID[2]-m_instrument.onChipData.m_InstruPos[2])<0.01 AND
	ABS(m_instrument.onChipData.m_InstruPosRFID[3]-m_instrument.onChipData.m_InstruPos[3])<0.01 THEN
	
	g_informationVerificationPassed:=TRUE;
END_IF;
GVL_InstruTestUIVars.g_RFID_SN:=ULINT_TO_STRING(m_instrument.onChipData.m_InstruseriesNumRFID);
IF (LEN(GVL_InstruTestUIVars.g_RFID_SN)=10)THEN
	GVL_InstruTestUIVars.g_RFID_SN:=concat('00',GVL_InstruTestUIVars.g_RFID_SN);
ELSIF  (LEN(GVL_InstruTestUIVars.g_RFID_SN)=11)THEN
	GVL_InstruTestUIVars.g_RFID_SN:=concat('0',GVL_InstruTestUIVars.g_RFID_SN);
ELSE
	GVL_InstruTestUIVars.g_RFID_SN:=GVL_InstruTestUIVars.g_RFID_SN;
END_IF
GVL_InstruTestUIVars.m_RFIDTimes:=ULINT_TO_DINT(m_instrument.onChipData.m_InstruUsageCountsRFID);
GVL_InstruTestUIVars.m_Instrument_pos_L1:=m_instrument.onChipData.m_InstruPosRFID[1];
GVL_InstruTestUIVars.m_Instrument_pos_L2:=m_instrument.onChipData.m_InstruPosRFID[2];
GVL_InstruTestUIVars.m_Instrument_pos_L3:=m_instrument.onChipData.m_InstruPosRFID[3];
GVL_InstruTestUIVars.g_informationVerificationPassed:=g_informationVerificationPassed;
GVL_InstruTestUIVars.g_readedRFID:=m_instrument.onChipData.m_InstruReadSucceedRFID;
IF GVL_InstruTestUIVars.g_readRFID AND iStepRFID=0 THEN
	GVL_InstruTestUIVars.g_readRFID:=FALSE;
	g_readedRFID:=FALSE;
	GVL_InstruTestUIVars.g_readRFIDFlag:=FALSE;
	uiRFIDReadSN:=0;
	iStepRFID:=3;
	iStepRFIDOnLine:=0;
END_IF
IF GVL_InstruTestUIVars.g_writeRFID AND iStepRFID=0 THEN
	GVL_InstruTestUIVars.g_writeRFID:=FALSE;
	iStepRFID:=53;
	iStepRFIDOnLine:=0;
END_IF

fbTonRFID(IN:=iStepRFID=10 OR iStepRFID=60, PT:=T#5S , Q=> , ET=> );
fbTonRFIDOnLine(IN:=m_offLineRFID , PT:=T#2S , Q=> , ET=> );
fbTonRFIDOnLineStep(IN:=iStepRFIDOnLine=10 , PT:=T#1S , Q=> , ET=> );
fbTonReadData(IN:=iStepRFID=15 OR iStepRFID=65 , PT:=T#0.5S , Q=> , ET=> );
IF fbTonRFIDOnLine.Q THEN
    g_offLineRFID:=FALSE;;
END_IF

CASE iStepRFID OF
	0:
(*		CASE iStepRFIDOnLine OF   //On  Off line
			0:
			  arrReadData:=arrRFIDData;
			  arrSendData:=arrRFIDData;
			  iStepRFIDOnLine:=5;
			5:   
			  arrSendData[1]:=16#FF;
			  arrSendData[2]:=16#08;  arrSendData[3]:=16#11;
			  arrSendData[4]:=16#00;  arrSendData[5]:=16#01;
			  arrSendData[6]:=16#00;  arrSendData[7]:=16#00;
			  arrSendData[8]:=16#01;  arrSendData[9]:=16#EF;
			  arrSendData[10]:=16#7F;  arrSendData[11]:=16#32;
			  bSend:=TRUE; 
			  iStepRFIDOnLine:=10;
			10:
			  IF arrReadData[0]<>0  THEN
				  g_offLineRFID:=TRUE;
				  m_offLineRFID:=FALSE;
			  ELSE
                  m_offLineRFID:=TRUE;
			  END_IF
			  IF fbTonRFIDOnLineStep.Q THEN
			  	  iStepRFIDOnLine:=0;
			  END_IF
		END_CASE
		
	*)	
    3:                           //Read
	  arrReadData:=arrRFIDData;
	  arrSendData:=arrRFIDData;
	  iStepRFID:=5;
	5:
	  arrSendData[0]:=16#FF;
	  arrSendData[1]:=16#08;  arrSendData[2]:=16#11;
	  arrSendData[3]:=16#00;  arrSendData[4]:=16#01;
	  arrSendData[5]:=16#00;  arrSendData[6]:=16#00;
	  arrSendData[7]:=16#01;  arrSendData[8]:=16#6E;
	  arrSendData[9]:=16#1F;  arrSendData[10]:=16#F2;
	  arrSendData[11]:=16#00; 
	  bSend:=TRUE; 
	  iStepRFID:=10;
	10:
	   IF arrReadData[0]<>0  THEN
		   iStepRFID:=15;
	   END_IF
	   IF fbTonRFID.Q THEN
		   iStepRFID:=0;
	       iStepRFIDOnLine:=0;
	   END_IF
	15: 
	IF fbTonReadData.Q THEN
//	   IF arrReadData[5]=0 THEN
	   	   iStepRFID:=20;
//	   END_IF
//	   IF arrReadData[5]<>0THEN
//	   	   iStepRFID:=30;
//	   END_IF
	END_IF
    20:
	   uiRFIDRead:=0;
	   FOR i:=8 TO 108 BY 1 DO
		    uiRFIDRead:=BYTE_TO_UINT(arrReadData[i])+uiRFIDRead;
	   END_FOR
  	   iStepRFID:=25;
	 25:
//	   AryByteTo(In:=arrReadData[111] , Size:= 2, Order:=_eBYTE_ORDER._HIGH_LOW , OutVal:=wCRCReadSum );
	   wCRCReadSum:=SHL(BYTE_TO_ULINT(arrReadData[109]),8)OR BYTE_TO_ULINT(arrReadData[110]);
	   IF wCRCReadSum=uiRFIDRead THEN
	    	g_readedRFID:=TRUE;
			GVL_InstruTestUIVars.g_readRFIDFlag:=TRUE;
			uiRFIDReadSN:=0;
	   FOR i:=1 TO 8 BY 1 DO
		  uiRFIDReadSN:=SHL(BYTE_TO_ULINT(arrReadData[58+i]),64-i*8)+uiRFIDReadSN;
	  END_FOR
	  m_readRFIDTimes:=0;
	   FOR i:=1 TO 4 BY 1 DO
		  m_readRFIDTimes:=SHL(BYTE_TO_DINT(arrReadData[68+i]),32-i*8)+m_readRFIDTimes;
	  END_FOR
	  m_readInstrument_pos_L1:=0;
	  m_readInstrument_pos_L2:=0;
	  m_readInstrument_pos_L3:=0;
	   FOR i:=1 TO 4 BY 1 DO
		  m_readInstrument_pos_L1:=DINT_TO_LREAL(SHL(BYTE_TO_DINT(arrReadData[28+i]),32-i*8))/1000+m_readInstrument_pos_L1;
	  END_FOR
	   FOR i:=1 TO 4 BY 1 DO
		  m_readInstrument_pos_L2:=DINT_TO_LREAL(SHL(BYTE_TO_DINT(arrReadData[38+i]),32-i*8))/1000+m_readInstrument_pos_L2;
	  END_FOR
	   FOR i:=1 TO 4 BY 1 DO
		  m_readInstrument_pos_L3:=DINT_TO_LREAL(SHL(BYTE_TO_DINT(arrReadData[48+i]),32-i*8))/1000+m_readInstrument_pos_L3;
	  END_FOR
	  
//			AryByteTo(In:=arrReadData[61] , Size:= 12, Order:=_eBYTE_ORDER._HIGH_LOW , OutVal:=uiRFIDReadSN );
//			m_instruPurpose:=BYTE_TO_INT(arrReadData[74]);
//			AryByteTo(In:=arrReadData[47] , Size:= 2, Order:=_eBYTE_ORDER._HIGH_LOW , OutVal:=m_maxClosingCurrent );
//			AryByteTo(In:=arrReadData[76] , Size:= 4, Order:=_eBYTE_ORDER._HIGH_LOW , OutVal:=m_readRFIDPos );
	    	iStepRFID:=0;
			iStepRFIDOnLine:=0;
	   ELSE
	        iStepRFID:=30;
	   END_IF
	 30:
	    g_readedRFID:=FALSE;
		GVL_InstruTestUIVars.g_readRFIDFlag:=FALSE;
	    iStepRFID:=0;
		iStepRFIDOnLine:=0;
 	 53:	                   //Write
	  arrReadData:=arrRFIDData;
	  arrSendData:=arrRFIDData;
	  iStepRFID:=55;
     55:  
	  arrSendData[0]:=16#FF;
	  arrSendData[1]:=16#76;  arrSendData[2]:=16#12;
	  arrSendData[3]:=16#00;  arrSendData[4]:=16#01;
	  arrSendData[5]:=16#00;  arrSendData[6]:=16#00;
	  arrSendData[7]:=16#00;  arrSendData[8]:=16#6E;  //Length  //110 BYTE
	  
	//  g_RFIDinstruSN:=g_newInstruSN;
	  //Data
	  arrSendData[11]:=(INT_TO_BYTE(g_moveMode) AND 16#0F) +(INT_TO_BYTE(SHL(g_energyType,4)) AND 16#F0);
	   FOR i:=1 TO 8 BY 1 DO
		  arrSendData[61+i]:=ULINT_TO_BYTE(SHR(g_RFIDinstruSN,64-i*8) );
	  END_FOR
	   FOR i:=1 TO 4 BY 1 DO
		  arrSendData[71+i]:=DINT_TO_BYTE(SHR(m_writeRFIDTimes,32-i*8) );
	  END_FOR
	   FOR i:=1 TO 4 BY 1 DO
		  arrSendData[31+i]:=DINT_TO_BYTE(SHR(LREAL_TO_DINT(m_writeInstrument_pos_L1*1000),32-i*8) );
	  END_FOR
	   FOR i:=1 TO 4 BY 1 DO
		  arrSendData[41+i]:=DINT_TO_BYTE(SHR(LREAL_TO_DINT(m_writeInstrument_pos_L2*1000),32-i*8) );
	  END_FOR
	   FOR i:=1 TO 4 BY 1 DO
		  arrSendData[51+i]:=DINT_TO_BYTE(SHR(LREAL_TO_DINT(m_writeInstrument_pos_L3*1000),32-i*8) );
	  END_FOR
	  
	   uiRFIDWrite:=0;  
	  FOR i:=11 TO 111 BY 1 DO                            //Sum 
		   uiRFIDWrite:=BYTE_TO_UINT(arrSendData[i])+uiRFIDWrite;
	  END_FOR
	  
	  arrSendData[112]:=UINT_TO_BYTE(SHR(uiRFIDWrite,8) );
	  arrSendData[113]:=UINT_TO_BYTE(uiRFIDWrite AND 16#00FF);
                   
	  wCRC16:=MEM.CRC16_Modbus(pMemoryBlock:= ADR(arrSendData ), uiLength:=119 );  //CRC
	  arrSendData[119]:=UINT_TO_BYTE(SHR(wCRC16,8) );
	  arrSendData[120]:=UINT_TO_BYTE(wCRC16 AND 16#00FF);
	  bSend:=TRUE; 
	  iStepRFID:=60;
	60:
	   IF arrReadData[0]<>0  THEN
           iStepRFID:=65;
	   END_IF
	   IF fbTonRFID.Q THEN
	   	   iStepRFID:=0;
		   iStepRFIDOnLine:=0;
	   END_IF
	65: 
	IF fbTonReadData.Q THEN
	   IF arrReadData[5]=0 THEN
	  	   iStepRFID:=75;
	   END_IF
	   IF arrReadData[5]<>0THEN
	   	   iStepRFID:=80;
	   END_IF
	END_IF
	 75:
	   g_writedRFID:=TRUE;
	   iStepRFID:=0;
	   iStepRFIDOnLine:=0;
	 80:
	   g_writedRFID:=FALSE;
	   iStepRFID:=0;
	   iStepRFIDOnLine:=0;
	  
END_CASE
	 (*
SNMid :=LREAL_TO_INT( FLOOR(ULINT_TO_LREAL(uiRFIDReadSN)/1000000000));
g_informationVerificationPassed:=FALSE;
IF g_readedRFID AND g_instruSN=uiRFIDReadSN  AND  (SNMid=042 OR SNMid=043 OR TRUE )AND 
	ABS(GVL_InstruTestUIVars.g_instruZeroPos[1]-m_readInstrument_pos_L1)<0.01 AND
	ABS(GVL_InstruTestUIVars.g_instruZeroPos[2]-m_readInstrument_pos_L2)<0.01 AND
	ABS(GVL_InstruTestUIVars.g_instruZeroPos[3]-m_readInstrument_pos_L3)<0.01 THEN
	
	g_informationVerificationPassed:=TRUE;
END_IF;

*)
IF g_informationVerificationPassed THEN
(*	g_instruPurposeUI:=m_instruPurpose;
	GVL_InstruTestUIVars.g_instruName:=1;
	GVL_InstruTestUIVars.g_numberOfUsableTimesUI:=1;
	GVL_InstruTestUIVars.g_usedTimesUI:=0;
	GVL_InstruTestUIVars.g_maxClosingCurrentUI:=m_maxClosingCurrent;
	IF SNMid=042 THEN
	    GVL_InstruTestUIVars.g_driveRodLengthUI:=464.6;
	    GVL_InstruTestUIVars.g_instruNameEnglish:=1;
		GVL_InstruTestUIVars.g_instruType:=1;
	ELSIF SNMid=043 THEN 
	    GVL_InstruTestUIVars.g_driveRodLengthUI:=552.3;
	    GVL_InstruTestUIVars.g_instruNameEnglish:=2;
		GVL_InstruTestUIVars.g_instruType:=2;
	END_IF
	GVL_InstruTestUIVars.g_maxWorkAngleUI:=45;
	GVL_InstruTestUIVars.g_reductionRatioK1UI:=25;
	GVL_InstruTestUIVars.g_reductionRatioK2UI:=13;
	GVL_InstruTestUIVars.g_reductionRatioK3UI:=18.5;
	GVL_InstruTestUIVars.g_moveModeUI:=5;
	GVL_InstruTestUIVars.g_energyTypeUI:=4;
	GVL_InstruTestUIVars.g_instruVersionUI:=01;
	GVL_InstruTestUIVars.g_formVersionUI:=01;
	GVL_InstruTestUIVars.g_readOpenAngleLinkPos:=DINT_TO_LREAL(m_readPos)/1000;
ELSE 
    GVL_InstruTestUIVars.g_instruPurposeUI:=0;
	GVL_InstruTestUIVars.g_instruName:=0;
	GVL_InstruTestUIVars.g_instruSN:=0;
	GVL_InstruTestUIVars.g_instruType:=0;
	GVL_InstruTestUIVars.g_numberOfUsableTimesUI:=0;
	GVL_InstruTestUIVars.g_usedTimesUI:=0;
	GVL_InstruTestUIVars.g_maxClosingCurrentUI:=0;
	GVL_InstruTestUIVars.g_driveRodLengthUI:=0;
	GVL_InstruTestUIVars.g_maxWorkAngleUI:=0;
	GVL_InstruTestUIVars.g_reductionRatioK1UI:=0;
	GVL_InstruTestUIVars.g_reductionRatioK2UI:=0;
	GVL_InstruTestUIVars.g_reductionRatioK3UI:=0;
	GVL_InstruTestUIVars.g_moveModeUI:=0;
	GVL_InstruTestUIVars.g_energyTypeUI:=0;
	GVL_InstruTestUIVars.g_instruVersionUI:=0;
	GVL_InstruTestUIVars.g_formVersionUI:=0;
	GVL_InstruTestUIVars.g_instruNameEnglish:=0;
	GVL_InstruTestUIVars.g_readOpenAngleLinkPos:=0;
	*)
END_IF
(*
IF m_instrument.onChipData.m_InstruReadSucceed THEN
	GVL_InstruTestUIVars.g_readSNNum:=m_instrument.onChipData.m_InstruseriesNum;
END_IF
GVL_InstruTestUIVars.g_readRFIDFlag:=g_readedRFID;
GVL_InstruTestUIVars.g_offLineRFID:=g_offLineRFID;
GVL_InstruTestUIVars.g_informationVerificationPassed:=g_informationVerificationPassed;
GVL_InstruTestUIVars.g_readedRFID:=g_readedRFID;
GVL_InstruTestUIVars.g_RFID_SN:=ULINT_TO_STRING(uiRFIDReadSN);
IF (LEN(GVL_InstruTestUIVars.g_RFID_SN)=10)THEN
	GVL_InstruTestUIVars.g_RFID_SN:=concat('00',GVL_InstruTestUIVars.g_RFID_SN);
ELSIF  (LEN(GVL_InstruTestUIVars.g_RFID_SN)=11)THEN
	GVL_InstruTestUIVars.g_RFID_SN:=concat('0',GVL_InstruTestUIVars.g_RFID_SN);
ELSE
	GVL_InstruTestUIVars.g_RFID_SN:=GVL_InstruTestUIVars.g_RFID_SN;
END_IF
IF m_instrument.onChipData.m_InstruReadSucceed THEN
	g_instruSN:= GVL_InstruTestUIVars.g_readSNNum;
	g_RFIDinstruSN:=GVL_InstruTestUIVars.g_readSNNum;
	m_writeRFIDTimes:=GVL_InstruTestUIVars.g_instruNumberOfUses;
	m_writeInstrument_pos_L1:=GVL_InstruTestUIVars.g_instruZeroPos[1];
	m_writeInstrument_pos_L2:=GVL_InstruTestUIVars.g_instruZeroPos[2];
	m_writeInstrument_pos_L3:=GVL_InstruTestUIVars.g_instruZeroPos[3];
END_IF
GVL_InstruTestUIVars.m_RFIDTimes:=m_readRFIDTimes;
GVL_InstruTestUIVars.m_Instrument_pos_L1:=m_readInstrument_pos_L1;
GVL_InstruTestUIVars.m_Instrument_pos_L2:=m_readInstrument_pos_L2;
GVL_InstruTestUIVars.m_Instrument_pos_L3:=m_readInstrument_pos_L3;
*)
(*
fbTonRFIDReaded(IN:=(GVL_InstruTestUIVars.IsolationPlate_Instrument_Install_Start AND 16#2)<>16#2,PT:=T#3S);
IF fbTonRFIDReaded.Q THEN
g_readedRFID:=FALSE;
END_IF
*)



//read recipe
IF (m_bReadRecipeStep<=2 AND m_bReadRecipeStep>0) THEN
	//The method loads a recipe from the specified recipe file.  It subsequently writes the recipe into the PLC variables.
    ReturnDwordRead:=RecipeManCommands.LoadAndWriteRecipe(RecipeDefinitionName:=GVL_SystemParameters.RecipeDefinitionName[m_bReadRecipeStep] , RecipeName:='RecipeRecord');
	IF ReturnDwordRead = ERR_OK THEN
		m_bReadRecipeStep:=m_bReadRecipeStep+1; 
	END_IF
END_IF 
//loadConfigFile := m_bReadRecipeStep>2;
//write recipe
IF m_saveAccount THEN	
	//This method creates a new recipe in the specified recipe definition. It subsequently reads the current PLC values into the new recipe and saves it as a recipe file with a standard name.
	 RecipeManCommands.CreateRecipe(RecipeDefinitionName:=GVL_SystemParameters.RecipeDefinitionName[1] , RecipeName:='RecipeRecord' );
	 ReturnDwordWrite:=RecipeManCommands.ReadAndSaveRecipe(RecipeDefinitionName:=GVL_SystemParameters.RecipeDefinitionName[1] , RecipeName:='RecipeRecord' ); 
	 m_saveAccount:=0;
END_IF
IF  m_saveCaliLinkEncoder THEN	
	//This method creates a new recipe in the specified recipe definition. It subsequently reads the current PLC values into the new recipe and saves it as a recipe file with a standard name.
	 RecipeManCommands.CreateRecipe(RecipeDefinitionName:=GVL_SystemParameters.RecipeDefinitionName[2] , RecipeName:='RecipeRecord' );
	 ReturnDwordWrite:=RecipeManCommands.ReadAndSaveRecipe(RecipeDefinitionName:=GVL_SystemParameters.RecipeDefinitionName[2] , RecipeName:='RecipeRecord' );
	 m_saveCaliLinkEncoder:=0;
END_IF

GVL_InstruTestUIVars.g_instruSNLen:=LEN(GVL_InstruTestUIVars.g_newInstruSN);
END_METHOD

METHOD checkLight : BOOL
VAR_INPUT
	i_lightCtrlWord : UDINT;
END_VAR

VAR
	lightCtrlWord : UDINT;
END_VAR
// to PDO
m_lightIO := UDINT_TO_DINT(i_lightCtrlWord);

// trig sdo write
lightCtrlWord := SHL(i_lightCtrlWord,16);
m_SdoWrite[1](sNetId:= m_armNetId, nSlaveAddr:= m_jointAddrJ8, nSubIndex:= 0, nIndex:= 16#6097, pSrcBuf:=ADR(lightCtrlWord) , cbBufLen:=SIZEOF(lightCtrlWord) , bExecute:= TRUE, tTimeout:= , bBusy=> , bError=> , nErrId=> );
m_SdoWrite[2](sNetId:= m_armNetId, nSlaveAddr:= m_jointAddrPbox, nSubIndex:= 0, nIndex:= 16#6097, pSrcBuf:= ADR(lightCtrlWord), cbBufLen:= SIZEOF(lightCtrlWord), bExecute:= TRUE, tTimeout:= , bBusy=> , bError=> , nErrId=> );

// disable sdo write
IF NOT m_SdoWrite[1].bBusy AND  NOT m_SdoWrite[2].bBusy THEN
	m_SdoWrite[1](bExecute:=FALSE);
	m_SdoWrite[2](bExecute:=FALSE);
END_IF
END_METHOD

PROPERTY cmdCartPose : REFERENCE TO ST_Frame
GET
cmdCartPose REF= m_cmdCartPose;
END_GET
END_PROPERTY

PROPERTY cmdCartTwist : REFERENCE to Vec6d
GET
cmdCartTwist REF= m_cmdCartTwist;
END_GET
END_PROPERTY

PROPERTY cmdJntCurrent : REFERENCE TO  Vec8d
GET
cmdJntCurrent ref= m_cmdJntCurrent;
END_GET
END_PROPERTY

PROPERTY cmdJntPos : REFERENCE TO Vec8d
GET
cmdJntPos REF= m_cmdJntPos;
END_GET
END_PROPERTY

PROPERTY cmdJntTrq :REFERENCE TO Vec8d
GET
cmdJntTrq REF= m_cmdJntTrq;
END_GET
END_PROPERTY

PROPERTY cmdJntVel : REFERENCE TO Vec8d
GET
cmdJntVel REF= m_cmdJntVel;
END_GET
END_PROPERTY

PROPERTY curCartPose : REFERENCE TO ST_Frame
GET
curCartPose ref=m_curCartPose;
END_GET
END_PROPERTY

PROPERTY curCartTwist : REFERENCE TO Vec6d
GET
curCartTwist ref=m_curCartTwist;
END_GET
END_PROPERTY

PROPERTY curDHJntPos :REFERENCE TO Vec6d
GET
curDHJntPos ref= m_curDHJntPos;
END_GET
END_PROPERTY

PROPERTY curDHJntVel :REFERENCE TO Vec6d
GET
curDHJntVel REF= m_curDHJntVel;
END_GET
END_PROPERTY

PROPERTY curGripAngle : LREAL
GET
curGripAngle:=m_curGripAngle;
END_GET
END_PROPERTY

PROPERTY curJntPos : REFERENCE TO Vec8d
GET
curJntPos ref=m_curJntPos;
END_GET
END_PROPERTY

PROPERTY curJntTrq : REFERENCE TO Vec8d
GET
curJntTrq ref=m_curJntTrq;
END_GET
END_PROPERTY

PROPERTY curJntVel :REFERENCE TO Vec8d
GET
curJntVel ref=m_curJntVel;
END_GET
END_PROPERTY

PROPERTY curLinkPos :REFERENCE TO Vec8d
GET
curLinkPos ref=m_curLinkPos;
END_GET
END_PROPERTY

PROPERTY curMotorPos : REFERENCE TO  Vec8d
GET
curMotorPos ref=m_curMotorPos;
END_GET
END_PROPERTY

METHOD PUBLIC enable : BOOL
VAR_IN_OUT CONSTANT
	i_jntIdx :Vec8i;
END_VAR
VAR
	i :INT ;
END_VAR
FOR i:=1 TO g_sJntNum DO
	IF 1= i_jntIdx[i] THEN
		m_joints[i].enable();
	ELSE
		m_joints[i].disable();
	END_IF
END_FOR
END_METHOD

PROPERTY filtJntCurrent :REFERENCE TO Vec8d
GET
filtJntCurrent ref= m_filtJntCurrent;
END_GET
END_PROPERTY

// from active joint position to cartesian pose in arm origin
METHOD PROTECTED forwardKinematic : BOOL
VAR_IN_OUT CONSTANT
	i_DHJntPos :Vec6d;
END_VAR
VAR_IN_OUT
	r_cartPose :ST_Frame;
END_VAR
VAR
	d1, L, a, b :LREAL;
	q3 :LREAL;

	c1,c2,c4,c5,c6,c7 :LREAL;
	s1,s2,s4,s5,s6,s7 :LREAL;
	DHRot :Mat3d;
	
	tmpRot1,tmpRot2 : Mat3d;

END_VAR

d1:=GVL_SlaveArmKinematic.g_d1;
L:=m_instrument.instruTypeInfo.m_rodLength;
a:=m_instrument.instruTypeInfo.m_headLength;
b:=m_instrument.instruTypeInfo.m_fingerLength;

q3:=i_DHJntPos[3];
c1:=COS(i_DHJntPos[1]);
c2:=COS(i_DHJntPos[2]);
c4:=COS(i_DHJntPos[4]);
c5:=COS(i_DHJntPos[5]);
c6:=COS(i_DHJntPos[6]);

s1:=SIN(i_DHJntPos[1]);
s2:=SIN(i_DHJntPos[2]);
s4:=SIN(i_DHJntPos[4]);
s5:=SIN(i_DHJntPos[5]);
s6:=SIN(i_DHJntPos[6]);


// cartesian pose frame
r_cartPose.m_pos[1]:=a*(c5*(s1*s4 + c1*c2*c4) - c1*s2*s5) + b*(c6*(c5*(s1*s4 + c1*c2*c4) - c1*s2*s5) - s6*(c4*s1 - c1*c2*s4)) + L*c1*s2 - q3*c1*s2;
r_cartPose.m_pos[2]:=a*(c2*s5 + c4*c5*s2) - d1 - L*c2 + q3*c2 + b*(c6*(c2*s5 + c4*c5*s2) + s2*s4*s6);
r_cartPose.m_pos[3]:=L*s1*s2 - a*(c5*(c1*s4 - c2*c4*s1) + s1*s2*s5) - b*(c6*(c5*(c1*s4 - c2*c4*s1) + s1*s2*s5) - s6*(c1*c4 + c2*s1*s4)) - q3*s1*s2;

DHRot[1,1]:= c6*(c5*(s1*s4 + c1*c2*c4) - c1*s2*s5) - s6*(c4*s1 - c1*c2*s4);
DHRot[2,1]:=c6*(c2*s5 + c4*c5*s2) + s2*s4*s6;
DHRot[3,1]:=s6*(c1*c4 + c2*s1*s4) - c6*(c5*(c1*s4 - c2*c4*s1) + s1*s2*s5);

DHRot[1,2]:=- s6*(c5*(s1*s4 + c1*c2*c4) - c1*s2*s5) - c6*(c4*s1 - c1*c2*s4);
DHRot[2,2]:=c6*s2*s4 - s6*(c2*s5 + c4*c5*s2);
DHRot[3,2]:=s6*(c5*(c1*s4 - c2*c4*s1) + s1*s2*s5) + c6*(c1*c4 + c2*s1*s4);

DHRot[1,3]:= s5*(s1*s4 + c1*c2*c4) + c1*c5*s2;
DHRot[2,3]:= c4*s2*s5 - c2*c5;
DHRot[3,3]:=c5*s1*s2 - s5*(c1*s4 - c2*c4*s1);

// convert to tcp rotation
matMultiply(DHRot, GVL_SlaveArmKinematic.g_tcpRotation, r_cartPOSE.m_rot);

//TODO: need verify
// rotate tcp coordinate 180 degree about z axis if instrument is a head-up 30deg endoscope
IF m_instrument.instruType = InstruType_Endoscope AND m_instrument.curScopeType = EndoScopeType_30 AND m_instrument.curScopePosture = EndoscopePosture_HeadUp THEN
	tmpRot2 := rotZ(pi);
	tmpRot1 := r_cartPOSE.m_rot;
	matMultiply(tmpRot1, tmpRot2, r_cartPOSE.m_rot);
END_IF
END_METHOD

METHOD PUBLIC init : BOOL
VAR_INPUT
	i_armIdx:INT;
END_VAR
VAR 
	i :INT ;
	currentRatioMotor2Jnt: LREAL;
END_VAR
// arm statues init
m_armIdx:=i_armIdx;
m_curGripAngle:=0;
m_simGripAngle:=0;

// joint init
FOR i:=1 TO g_sJntNum DO
	IF i<4 THEN
		m_joints[i].init(m_armIdx, i,g_slaveArmCtrlCycleTime, 1);
	ELSE
		m_joints[i].init(m_armIdx, i,g_slaveArmCtrlCycleTime, 4);
	END_IF
END_FOR

// init joint encoder and position calculation
initJntPos();

// joint controller init
FOR i:=1 TO g_sJntNum DO 
	currentRatioMotor2Jnt:=GVL_SlaveMotorParameters.g_motorTrqConst[i]*GVL_SlaveMotorParameters.g_motorReduction[i]/1000;
	m_jntPIDCtrl[i].init(g_slaveArmCtrlCycleTime,GVL_slaveControlParameters.g_posKp[i],GVL_slaveControlParameters.g_posKd[i],
		GVL_slaveControlParameters.g_posKi[i], GVL_slaveControlParameters.g_posKiLimit[i]* currentRatioMotor2Jnt,
		GVL_slaveControlParameters.g_posCtrlLimit[i]*currentRatioMotor2Jnt);
END_FOR

// instrument init
m_instrument.init(i_armIdx);

//init arm netID and adrr
m_armNetId := GVL_SlaveJointEncoderCaliData.g_slaveArmNetID[armIdx];
m_jointAddrJ8 := GVL_SlaveJointEncoderCaliData.g_slaveJointNetPort[armIdx,3];
m_jointAddrPbox := GVL_SlaveJointEncoderCaliData.g_slaveJointNetPort[armIdx,4];

// endosocpe toggle button check
m_endoscopeTypeSwitch.init(0, 500);
m_endoscopePostureSwitch.init(0,500);
END_METHOD

METHOD PUBLIC initJntPos : BOOL
VAR_INPUT
END_VAR
VAR
	i:INT ;
END_VAR
// joint init
FOR i:=1 TO g_sJntNum DO
	m_joints[i].initJntPos();
END_FOR

// update arm status if joint position is re-init
updateStatus();
END_METHOD

PROPERTY instrument : REFERENCE TO FB_Instrument
GET
instrument REF=m_instrument;
END_GET
END_PROPERTY

PROPERTY instruNear : BOOL
GET
instruNear := m_instruNearFlag;
END_GET
END_PROPERTY

PROPERTY instruOn : bool
GET
instruOn:=m_instruOnFlag;
END_GET
END_PROPERTY

// check if instrument is in ready position(far enough from romote center) for following manipulation
METHOD PUBLIC instruReady : BOOL
VAR_INPUT
END_VAR

VAR
	// check buffer
	checkBuffer :LREAL := 0.005;
END_VAR
IF NOT(m_instrument.onChipData.m_InstruReadSucceed) THEN
	instruReady :=FALSE;
	RETURN;
END_IF

instruReady := m_curJntPos[3] < (m_instrument.instruTypeInfo.m_rodLength+m_instrument.instruTypeInfo.m_headLength
									+ m_instrument.instruTypeInfo.m_fingerLength - GVL_SlaveArmKinematic.g_minInstruRCDis+checkBuffer);
END_METHOD

METHOD PUBLIC isEnabled : BOOL
VAR_IN_OUT CONSTANT
	i_jntIdx :Vec8i;
END_VAR
VAR
	i :INT ;
END_VAR
isEnabled := TRUE;
FOR i:=1 TO g_sJntNum DO
	IF 1= i_jntIdx[i] THEN
		isEnabled :=  (m_joints[i].isEnabled() AND isEnabled);
	END_IF
END_FOR
END_METHOD

PROPERTY isSingurality : bool
GET
isSingurality:=m_isSingularity;
END_GET
END_PROPERTY

PROPERTY jaco :REFERENCE TO Mat6d
GET
jaco ref= m_jaco;
END_GET
END_PROPERTY

PROPERTY jntGravity :REFERENCE TO Vec8d
GET
jntGravity ref=m_jntGravity;
END_GET
END_PROPERTY

PROPERTY linkSingle : REFERENCE TO Vec8d
GET
linkSingle ref=m_curLinkSingle;
END_GET
END_PROPERTY

PROPERTY PUBLIC massMat :REFERENCE TO Mat3d
GET
massMat ref=m_jntMassMat;
END_GET
END_PROPERTY

METHOD mes : BOOL
VAR_INPUT
END_VAR
GVL_MES.g_serialNumLen:=LEN(GVL_MES.g_serialNum);
IF GVL_MES.g_serialNum<>m_serialNumOld AND GVL_MES.g_serialNumLen=9 THEN
	GVL_MES.g_eventTime[1]:=m_time;
END_IF
m_serialNumOld:=GVL_MES.g_serialNum;
GVL_MES.g_actualAccountNumber:=GVL_InstruTestUIVars.g_account.actualAccountNumber;
IF m_logStep=15 THEN
	GVL_MES.g_eventTime[2]:=m_time;
END_IF
GVL_MES.g_powerBoxCalibrationPos:=GVL_SlaveJointEncoderCaliData.g_caliLinkEncoder;
IF GVL_InstruTestUIVars.g_powerBoxCalibrationFlag=FALSE THEN
	GVL_MES.g_eventTime[3]:=m_time;
END_IF
GVL_MES.g_SN:=GVL_InstruTestUIVars.g_instruSN;
IF startFlag THEN
	GVL_MES.g_eventTime[4]:=m_time;
END_IF
GVL_MES.g_writeInstruZeroPos:=GVL_InstruTestUIVars.writeInstruZeroPos;
IF GVL_InstruTestUIVars.g_writeZeroPosFlag THEN
	GVL_MES.g_eventTime[5]:=m_time;
END_IF
GVL_MES.g_instruZeroPos:=GVL_InstruTestUIVars.g_instruZeroPos;
IF startFlag THEN
	GVL_MES.g_eventTime[6]:=m_time;
END_IF
GVL_MES.g_readRFIDFlig:=g_readedRFID;
IF iStepRFID=5 THEN
	GVL_MES.g_eventTime[7]:=m_time;
END_IF
IF GVL_MES.g_autoTestMode=3 OR GVL_MES.g_autoTestMode=13 THEN
	GVL_MES.g_curNumTiredTest:=GVL_InstruTestUIVars.g_curTestCycles;
ELSE
	GVL_MES.g_curNumTiredTest:=0;
END_IF
IF m_curTestCyclesOld<>GVL_InstruTestUIVars.g_curTestCycles AND(GVL_MES.g_autoTestMode=3 OR GVL_MES.g_autoTestMode=13) THEN
	GVL_MES.g_eventTime[8]:=m_time;
END_IF
m_curTestCyclesOld:=GVL_InstruTestUIVars.g_curTestCycles;
IF GVL_MES.g_attitudeOK THEN
	GVL_MES.g_attitudeConfirm:=1;
	GVL_MES.g_attitudeOK:=0;
	GVL_MES.g_eventTime[9]:=m_time;
ELSIF
	GVL_MES.g_attitudeNG THEN
	GVL_MES.g_attitudeConfirm:=2;
	GVL_MES.g_attitudeNG:=0;
	GVL_MES.g_eventTime[9]:=m_time;
END_IF
END_METHOD

METHOD PROTECTED modifyJaco : BOOL
VAR_IN_OUT CONSTANT
	i_DHJntPos :Vec6d;
END_VAR
VAR_IN_OUT
	r_jaco :Mat6d;
END_VAR

VAR CONSTANT
	// modify joint2/3 position to avoid jacobian singularity
	m_Jnt2PosThres :LREAL := -165 * g_deg2Rad;
	m_Jnt3PosThres :LREAL := -0.03;
END_VAR

VAR
	d1, L, a, b :LREAL;
	q2, q3:LREAL;

	c1,c2,c4,c5,c6,c7 :LREAL;
	s1,s2,s4,s5,s6,s7 :LREAL;
END_VAR
d1:=GVL_SlaveArmKinematic.g_d1;
L:=m_instrument.instruTypeInfo.m_rodLength;
a:=m_instrument.instruTypeInfo.m_headLength;
b:=m_instrument.instruTypeInfo.m_fingerLength;

q2 := i_DHJntPos[2];
IF q2 < m_Jnt2PosThres THEN
	q2 := m_Jnt2PosThres;
END_IF

q3:=i_DHJntPos[3];
IF q3 - L > m_Jnt3PosThres THEN
	q3:= L + m_Jnt3PosThres;
END_IF

c1:=COS(i_DHJntPos[1]);
c2:=COS(q2);
c4:=COS(i_DHJntPos[4]);
c5:=COS(i_DHJntPos[5]);
c6:=COS(i_DHJntPos[6]);

s1:=SIN(i_DHJntPos[1]);
s2:=SIN(q2);
s4:=SIN(i_DHJntPos[4]);
s5:=SIN(i_DHJntPos[5]);
s6:=SIN(i_DHJntPos[6]);

// jacobian with DH joints
r_jaco[1,1]:=b*(c6*(c5*(c1*s4 - c2*c4*s1) + s1*s2*s5) - s6*(c1*c4 + c2*s1*s4)) + a*(c5*(c1*s4 - c2*c4*s1) + s1*s2*s5) - L*s1*s2 + q3*s1*s2;
r_jaco[1,2]:=-c1*(a*(c2*s5 + c4*c5*s2) - L*c2 + q3*c2 + b*(c6*(c2*s5 + c4*c5*s2) + s2*s4*s6));
r_jaco[1,3]:=-c1*s2;
r_jaco[1,4]:=s1*s2*(a*(c2*s5 + c4*c5*s2) + b*(c6*(c2*s5 + c4*c5*s2) + s2*s4*s6)) - c2*(b*(c6*(c5*(c1*s4 - c2*c4*s1) + s1*s2*s5) - s6*(c1*c4 + c2*s1*s4)) + a*(c5*(c1*s4 - c2*c4*s1) + s1*s2*s5));
r_jaco[1,5]:=- (a*(c2*s5 + c4*c5*s2) + b*(c6*(c2*s5 + c4*c5*s2) + s2*s4*s6))*(c1*c4 + c2*s1*s4) - s2*s4*(b*(c6*(c5*(c1*s4 - c2*c4*s1) + s1*s2*s5) - s6*(c1*c4 + c2*s1*s4)) + a*(c5*(c1*s4 - c2*c4*s1) + s1*s2*s5));
r_jaco[1,6]:= b*(c6*(c5*(c1*s4 - c2*c4*s1) + s1*s2*s5) - s6*(c1*c4 + c2*s1*s4))*(c2*c5 - c4*s2*s5) + b*(s5*(c1*s4 - c2*c4*s1) - c5*s1*s2)*(c6*(c2*s5 + c4*c5*s2) + s2*s4*s6);


r_jaco[2,1]:=0;
r_jaco[2,2]:=c1*(a*(c5*(s1*s4 + c1*c2*c4) - c1*s2*s5) + b*(c6*(c5*(s1*s4 + c1*c2*c4) - c1*s2*s5) - s6*(c4*s1 - c1*c2*s4)) + L*c1*s2 - q3*c1*s2) - s1*(b*(c6*(c5*(c1*s4 - c2*c4*s1) + s1*s2*s5) - s6*(c1*c4 + c2*s1*s4)) + a*(c5*(c1*s4 - c2*c4*s1) + s1*s2*s5) - L*s1*s2 + q3*s1*s2);
r_jaco[2,3]:= c2;
r_jaco[2,4]:=- s1*s2*(a*(c5*(s1*s4 + c1*c2*c4) - c1*s2*s5) + b*(c6*(c5*(s1*s4 + c1*c2*c4) - c1*s2*s5) - s6*(c4*s1 - c1*c2*s4))) - c1*s2*(b*(c6*(c5*(c1*s4 - c2*c4*s1) + s1*s2*s5) - s6*(c1*c4 + c2*s1*s4)) + a*(c5*(c1*s4 - c2*c4*s1) + s1*s2*s5));
r_jaco[2,5]:=(a*(c5*(s1*s4 + c1*c2*c4) - c1*s2*s5) + b*(c6*(c5*(s1*s4 + c1*c2*c4) - c1*s2*s5) - s6*(c4*s1 - c1*c2*s4)))*(c1*c4 + c2*s1*s4) - (b*(c6*(c5*(c1*s4 - c2*c4*s1) + s1*s2*s5) - s6*(c1*c4 + c2*s1*s4)) + a*(c5*(c1*s4 - c2*c4*s1) + s1*s2*s5))*(c4*s1 - c1*c2*s4);
r_jaco[2,6]:=b*(c6*(c5*(c1*s4 - c2*c4*s1) + s1*s2*s5) - s6*(c1*c4 + c2*s1*s4))*(s5*(s1*s4 + c1*c2*c4) + c1*c5*s2) - b*(s5*(c1*s4 - c2*c4*s1) - c5*s1*s2)*(c6*(c5*(s1*s4 + c1*c2*c4) - c1*s2*s5) - s6*(c4*s1 - c1*c2*s4));

r_jaco[3,1]:=a*(c5*(s1*s4 + c1*c2*c4) - c1*s2*s5) + b*(c6*(c5*(s1*s4 + c1*c2*c4) - c1*s2*s5) - s6*(c4*s1 - c1*c2*s4)) + L*c1*s2 - q3*c1*s2;
r_jaco[3,2]:=-s1*(a*(c2*s5 + c4*c5*s2) - L*c2 + q3*c2 + b*(c6*(c2*s5 + c4*c5*s2) + s2*s4*s6));
r_jaco[3,3]:=-s1*s2;
r_jaco[3,4]:=- c2*(a*(c5*(s1*s4 + c1*c2*c4) - c1*s2*s5) + b*(c6*(c5*(s1*s4 + c1*c2*c4) - c1*s2*s5) - s6*(c4*s1 - c1*c2*s4))) - c1*s2*(a*(c2*s5 + c4*c5*s2) + b*(c6*(c2*s5 + c4*c5*s2) + s2*s4*s6));
r_jaco[3,5]:=- (a*(c2*s5 + c4*c5*s2) + b*(c6*(c2*s5 + c4*c5*s2) + s2*s4*s6))*(c4*s1 - c1*c2*s4) - s2*s4*(a*(c5*(s1*s4 + c1*c2*c4) - c1*s2*s5) + b*(c6*(c5*(s1*s4 + c1*c2*c4) - c1*s2*s5) - s6*(c4*s1 - c1*c2*s4)));
r_jaco[3,6]:=b*(c6*(c5*(s1*s4 + c1*c2*c4) - c1*s2*s5) - s6*(c4*s1 - c1*c2*s4))*(c2*c5 - c4*s2*s5) + b*(c6*(c2*s5 + c4*c5*s2) + s2*s4*s6)*(s5*(s1*s4 + c1*c2*c4) + c1*c5*s2);

r_jaco[4,1]:=0;
r_jaco[4,2]:=-s1;
r_jaco[4,3]:=0;
r_jaco[4,4]:=-c1*s2;
r_jaco[4,5]:=c1*c2*s4 - c4*s1;
r_jaco[4,6]:=s5*(s1*s4 + c1*c2*c4) + c1*c5*s2;

r_jaco[5,1]:=-1;
r_jaco[5,2]:=0;
r_jaco[5,3]:=0;
r_jaco[5,4]:=c2;
r_jaco[5,5]:=s2*s4;
r_jaco[5,6]:=c4*s2*s5 - c2*c5;

r_jaco[6,1]:=0;
r_jaco[6,2]:=c1;
r_jaco[6,3]:=0;
r_jaco[6,4]:=-s1*s2;
r_jaco[6,5]:=c1*c4 + c2*s1*s4;
r_jaco[6,6]:=c5*s1*s2 - s5*(c1*s4 - c2*c4*s1);
END_METHOD

PROPERTY panelOn : bool
GET
panelOn :=m_panelOnFlag;
END_GET
END_PROPERTY

PROPERTY rawJntCurrent :REFERENCE TO Vec8d
GET
rawJntCurrent ref=m_rawJntCurrent;
END_GET
END_PROPERTY

// check if instrument is in ready position(far enough from romote center) for following manipulation
METHOD PUBLIC readyForInstruMount : BOOL
VAR_INPUT
END_VAR

VAR
	// check buffer
	checkBuffer :LREAL := 0.01;
END_VAR
readyForInstruMount := (m_curJntPos[3]> GVL_SlaveMotorParameters.g_maxDHJntPos[3]-checkBuffer AND m_panelOnFlag);
END_METHOD

METHOD PUBLIC resetInstruDepth : BOOL
VAR_INPUT
END_VAR
m_instruInvasionDepth :=GVL_SlaveMotorParameters.g_maxJntPos[3];
END_METHOD

METHOD PUBLIC setInstruDepth : BOOL
VAR_INPUT
END_VAR
m_instruInvasionDepth := m_curJntPos[3]-m_instrument.instruTypeInfo.m_rodLength-m_instrument.instruTypeInfo.m_headLength
						- m_instrument.instruTypeInfo.m_fingerLength;
END_METHOD

METHOD setSaveCaliLinkEncoder : BOOL
VAR_INPUT
END_VAR
m_saveCaliLinkEncoder:=1;
END_METHOD

PROPERTY simCartPose :REFERENCE TO ST_Frame
GET
simCartPose ref=m_simCartPose;
END_GET
END_PROPERTY

PROPERTY simDHJntPos :REFERENCE TO Vec6d
GET
simDHJntPos ref= m_simDHJntPos;
END_GET
END_PROPERTY

PROPERTY simGripAngle : LREAL
GET
simGripAngle:=m_simGripAngle;
END_GET
END_PROPERTY

PROPERTY simJaco :REFERENCE TO mat6d
GET
simJaco ref=m_simJaco;
END_GET
END_PROPERTY

PROPERTY simJacoInv :REFERENCE TO Mat6d
GET
simJacoInv ref= m_simJacoInv;
END_GET
END_PROPERTY

PROPERTY PUBLIC trocarOn : bool
GET
trocarOn := m_trocarOnFlag;
END_GET
END_PROPERTY

// update joints control command
METHOD PUBLIC updateCmds : BOOL
VAR_IN_OUT CONSTANT
	i_armCtrlCmd : ST_SlaveArmCtrlCmds;
END_VAR
VAR
	i:INT;
END_VAR
m_cmdJntTrq:=i_armCtrlCmd.m_cmdJntTrq;
m_cmdJntPos :=i_armCtrlCmd.m_cmdJntPos;
m_cmdJntVel :=i_armCtrlCmd.m_cmdJntVel;
m_cmdCartTwist := i_armCtrlCmd.m_cmdCartTwist;
m_cmdCartPose :=i_armCtrlCmd.m_cmdCartPose;
m_simJntPos:=i_armCtrlCmd.m_simJntPos;

// update simulated master arm
updateSimStatus();

// enable/disable joints
enable(i_armCtrlCmd.m_jntEnableFlag);

m_codeTime(START:=TRUE, RESET:=TRUE);
// position/torque control
FOR i:=1 TO g_sJntNum DO 
	m_joints[i].setMaxCurrent(GVL_InstruTestUIVars.g_actualRatedCurrent[i]);
	IF i_armCtrlCmd.m_jntOPMode[i]=DriverOPMode_PosTrq THEN
		// position controller and gravity feedforward
		m_cmdJntTrq[i]:=m_jntPIDCtrl[i].run(m_cmdJntPos[i],m_curJntPos[i],m_cmdJntVel[i],m_curJntVel[i]);
		m_cmdJntTrq[i]:=m_cmdJntTrq[i]+m_jntGravity[i] + i_armCtrlCmd.m_FFJntTrq[i];
		m_joints[i].updateCmds(DriverOPMode_Trq,m_cmdJntPos[i],m_cmdJntTrq[i]);
	ELSIF i_armCtrlCmd.m_jntOPMode[i]=DriverOPMode_Trq THEN
		// gravity feedforward
		m_jntPIDCtrl[i].reset();
		m_cmdJntTrq[i]:=m_cmdJntTrq[i]+m_jntGravity[i];
		m_joints[i].updateCmds(DriverOPMode_Trq,m_cmdJntPos[i],m_cmdJntTrq[i]);
	ELSE
		m_jntPIDCtrl[i].reset();
		m_cmdJntTrq[i]:=0;
		m_joints[i].updateCmds(DriverOPMode_Pos,m_cmdJntPos[i],m_cmdJntTrq[i]);
	END_IF
	
END_FOR
m_codeTime(START:=FALSE);
END_METHOD

METHOD PUBLIC updateDyna : BOOL
VAR_IN_out constant
	slaveDynaData : ST_SlaveDynaData;
END_VAR
m_jntMassMat:=slaveDynaData.m_massMat[m_armIdx];
m_jntGravity[1]:=slaveDynaData.m_gravity[m_armIdx][1];
m_jntGravity[2]:=slaveDynaData.m_gravity[m_armIdx][2];
m_jntGravity[3]:=slaveDynaData.m_gravity[m_armIdx][3];
END_METHOD

METHOD PUBLIC updateSimStatus : BOOL
VAR_INPUT
END_VAR
//IF m_instrument.ready THEN
	// instrument kinematic
	m_instrument.instruFK(m_simJntPos, m_simDHJntPos, m_simGripAngle);

	// simulated cartesion pose 
	forwardKinematic(m_simDHJntPos,m_simCartPose);
	
	// simulated jacobian
	modifyJaco(m_simDHJntPos,m_simJaco);
	m_isSingularity:=NOT(invMat6(m_simJaco, m_simJacoInv));
//END_IF
END_METHOD

// update arm status, including kinematic and dynamic
METHOD PUBLIC updateStatus : BOOL
VAR_INPUT
END_VAR
VAR 
	i,j:INT;
END_VAR
// update joint data
FOR i:=1 TO g_sJntNum DO
	m_joints[i].updateStatus();
END_FOR

// check IO informantion
checkIO();

//mes
mes();

// get joint data
FOR i:=1 TO g_sJntNum DO
	m_curMotorPos[i]:=m_joints[i].motorPos;
	m_curLinkPos[i]:=m_joints[i].linkPos;
	m_curLinkSingle[i]:=m_joints[i].linkSingle;
	m_curJntPos[i]:=m_joints[i].jntPos;
	m_curJntVel[i]:=m_joints[i].jntVel;
	m_curJntTrq[i]:=m_joints[i].jntTrq;
	m_rawJntCurrent[i]:=m_joints[i].rawCurrent;
	m_filtJntCurrent[i]:=m_joints[i].filtCurrent;
	m_cmdJntCurrent[i]:=m_joints[i].cmdCurrent;
END_FOR 

// only update carteisn data when instrument is ready
//IF m_instrument.ready THEN
	
	// instrument kinematic
	m_instrument.instruFK(m_curJntPos, m_curDHJntPos, m_curGripAngle);

	// cartesion pose
	forwardKinematic(m_curDHJntPos,m_curCartPose);
	
	// jacobian
	calcJaco(m_curDHJntPos,m_jaco);
	
	// DH joint velocity
	m_instrument.instruJntVelFK(m_curJntVel, m_curDHJntVel);
	
	// cartesian twist
	matMultiVec(m_jaco, m_curDHJntVel, m_curCartTwist);
//END_IF
END_METHOD

END_FUNCTION_BLOCK

// ---- FBs_Robots/FB_SlaveJoint.TcPOU
FUNCTION_BLOCK FB_SlaveJoint EXTENDS FB_JointBase
VAR_INPUT
END_VAR
VAR_OUTPUT
END_VAR
VAR
	// power box joint motor rated current
	m_wristJntRatedCurrent : DINT := 540;

END_VAR

METHOD PUBLIC init : BOOL
VAR_INPUT
	i_armIdx :INT;
	i_jntIdx :INT;
	i_controlCycleTime :LREAL;
	// velocity is calculated every (m_velCalcCycles) control cycles
	// TODO: insturment joint motor can not reach 4k now, so calculate their velocity with 1k frequency, need to remove later
	i_velCalcCycles :INT;
END_VAR
m_armIdx:=i_armIdx;
m_jntIdx:=i_jntIdx;
m_cycleTime := i_controlCycleTime;
m_velCalcCycles :=MAX(i_velCalcCycles,1);

// hardware parameters
m_motorEncoderRes :=GVL_SlaveMotorParameters.g_incEncoderRes[i_jntIdx];
m_linkEncoderRes :=GVL_SlaveMotorParameters.g_absEncoderRes[i_jntIdx];
m_motorReduction :=GVL_SlaveMotorParameters.g_motorReduction[i_jntIdx];
m_linkEncoderReduction :=GVL_SlaveMotorParameters.g_absEncoderReduction[i_jntIdx];
m_trqConst :=GVL_SlaveMotorParameters.g_motorTrqConst[i_jntIdx];
m_maxCurrent :=GVL_SlaveMotorParameters.g_motorMaxCurrent[i_jntIdx];
m_motorDir :=GVL_SlaveMotorParameters.g_motorDir[i_jntIdx];								
m_minJntPos	:=GVL_SlaveMotorParameters.g_minJntPos[i_jntIdx];
m_maxJntPos	:=GVL_SlaveMotorParameters.g_maxJntPos[i_jntIdx];

//link encoder calibartion data
m_linkEncoderDir :=GVL_SlaveJointEncoderCaliData.g_asbEncoderDir[i_jntIdx];
m_minLinkEncoder :=GVL_SlaveJointEncoderCaliData.g_minLinkEncoder[i_armIdx, i_jntIdx] - m_linkEncoderDir*GVL_SlaveJointEncoderCaliData.g_linkEncLimitBuffer; // expand limit
m_maxLinkEncoder :=GVL_SlaveJointEncoderCaliData.g_maxLinkEncoder[i_armIdx, i_jntIdx] + m_linkEncoderDir*GVL_SlaveJointEncoderCaliData.g_linkEncLimitBuffer; // expand limit
m_caliLinkEncoder :=GVL_SlaveJointEncoderCaliData.g_caliLinkEncoder[i_armIdx, i_jntIdx];
m_linkEncCaliJntPos :=GVL_SlaveJointEncoderCaliData.g_linkEncCaliJntPos[i_jntIdx];
m_linkEncZeroCross :=GVL_SlaveJointEncoderCaliData.g_linkEncZeroCross[i_armIdx, i_jntIdx];
m_multiCycles :=GVL_SlaveJointEncoderCaliData.g_multipleCyclesJoint[i_armIdx,i_jntIdx];

// convert cali link encoder if joint cross zero
IF 1=m_linkEncZeroCross THEN
	IF 1=m_linkEncoderDir AND m_caliLinkEncoder < m_minLinkEncoder THEN
		m_caliLinkEncoder := GVL_SlaveJointEncoderCaliData.g_caliLinkEncoder[i_armIdx, i_jntIdx] + m_linkEncoderRes;
	ELSIF -1=m_linkEncoderDir AND m_caliLinkEncoder < m_maxLinkEncoder THEN
		m_caliLinkEncoder := GVL_SlaveJointEncoderCaliData.g_caliLinkEncoder[i_armIdx, i_jntIdx] + m_linkEncoderRes;
	END_IF
END_IF

// macro data
m_trq2CurrentRatio:=m_motorDir * 1000.0/(m_trqConst*m_motorReduction);
m_current2TrqRatio:=m_motorDir * (m_trqConst*m_motorReduction)/1000.0;
m_linkEnc2PosRatio := 2*PI*m_linkEncoderDir/(m_linkEncoderReduction*m_linkEncoderRes);
m_motorEnc2PosRatio := 2*PI * m_motorDir/(m_motorReduction * m_motorEncoderRes);

// motor data init
m_rawJntVel :=0;
m_curJntVel:=0;
m_curJntTrq :=0;
m_rawCurrent :=0;
m_filtCurrent :=0;
m_cmdJntVel :=0.0;
m_cmdJntTrq :=0.0;
m_cmdCurrent := 0.0;

// filter init
m_jntVelLpf.init(1, GVL_SlaveControlParameters.g_curJntVelLpfCutoffFreq, g_slaveArmCtrlFreq/m_velCalcCycles);
m_cmdTrqLpf.init(1, GVL_SlaveControlParameters.g_cmdJntTrqLpfCutoffFreq, g_slaveArmCtrlFreq);
m_curTrqLpf.init(1, GVL_SlaveControlParameters.g_curJntTrqLpfCutoffFreq, g_slaveArmCtrlFreq);

// driver init value
m_motorOutputs.m_controlWord:=DriverCtrlWord_INIT;
m_motorOutputs.m_opMode:=INT_TO_SINT(DriverOPMode_Pos);
m_motorOutputs.m_cmdCurrent:=0;
m_motorOutputs.m_cmdMotorEncoder:=m_motorInputs.m_motorEncoder;
END_METHOD

METHOD setMaxCurrent : BOOL
VAR_INPUT
	i_maxCurrent :LREAL;
END_VAR
m_maxCurrent := i_maxCurrent;
END_METHOD

METHOD PUBLIC updateCmds : BOOL
VAR_INPUT
	i_opMode : E_DriverOPMode;
	i_cmdPos :LREAL;
	i_cmdTrq :LREAL;
END_VAR
VAR
	filtCmdTrq :LREAL;
END_VAR
SUPER^.updateCmds(i_opMode, i_cmdPos, i_cmdTrq);

// write SDO data
writeSDOData();
END_METHOD

METHOD PROTECTED writeSDOData : BOOL
VAR_INPUT
END_VAR
VAR
	SDOSubIndexMode :WORD;
	SDOSubIndexCur :WORD;
END_VAR
//动力盒移动关节和器械旋转关节，共享一个控制字，由SDO写入
//IF (m_jntIdx=3) OR (m_jntIdx=8)  THEN
//	SDOSubIndexMode :=16#609B;
//	SDOSubIndexCur:=16#6098;
////动力盒3、5号电机为一个驱动器，共享一个控制字，由SDO写入
//ELSIF (m_jntIdx=4) OR (m_jntIdx=6)  THEN
//	SDOSubIndexMode :=16#609C;
//	SDOSubIndexCur:=16#6099;
////动力盒2、4号电机为一个驱动器，共享一个控制字，由SDO写入
//ELSIF (m_jntIdx=5) OR (m_jntIdx=7)  THEN
//	SDOSubIndexMode :=16#609D;
//	SDOSubIndexCur:=16#609A;
//END_IF
SDOSubIndexCur:=16#6090;
IF m_jntIdx <3 THEN
	RETURN;
END_IF

// write driver operation mode if it changs
//IF  m_jntIdx >=3 AND m_jntIdx <=8 THEN
//	m_opModeSDOWrite(sNetID:= GVL_SlaveJointEncoderCaliData.g_slaveArmNetID[m_armIdx],
//					nSlaveAddr := GVL_SlaveJointEncoderCaliData.g_slaveJointNetPort[m_armIdx,m_jntIdx],
//					nSubIndex:=0,nIndex:=SDOSubIndexMode,pSrcBuf:=ADR(m_motorOutputs.m_opMode),cbBufLen:=SIZEOF(m_motorOutputs.m_opMode),bExecute:=TRUE);
//	IF NOT m_opModeSDOWrite.bBusy THEN
//		m_opModeSDOWrite(bExecute:=FALSE);
//	END_IF
//END_IF
m_wristJntRatedCurrent := LREAL_TO_DINT(m_maxCurrent);
// write max motor current if it changes and works in position mode
IF m_jntIdx =4 OR m_jntIdx =6  THEN 
	m_MotorCurrentSDOWrite(sNetID:= GVL_SlaveJointEncoderCaliData.g_slaveArmNetID[m_armIdx],
					nSlaveAddr := GVL_SlaveJointEncoderCaliData.g_slaveJointNetPort[m_armIdx,m_jntIdx],
					nSubIndex:=06,nIndex:=SDOSubIndexCur,pSrcBuf:=ADR(m_wristJntRatedCurrent),cbBufLen:=SIZEOF(m_wristJntRatedCurrent),bExecute:=TRUE);
	IF NOT m_MotorCurrentSDOWrite.bBusy THEN
		m_MotorCurrentSDOWrite(bExecute:=FALSE);
	END_IF
END_IF
END_METHOD

END_FUNCTION_BLOCK

// ---- FBs_BasicControllers/FB_UltrosonicKnifeControl.TcPOU
// instrument joints control
FUNCTION_BLOCK FB_UltrosonicKnifeControl
VAR_INPUT
END_VAR
VAR_OUTPUT
END_VAR
VAR
	// instrument PID control paramters
	m_instruKp:ARRAY[1..5] OF LREAL:=[5(3)];
	m_instruKd:ARRAY[1..5] OF LREAL:=[5(0.04)];
	m_instruKi:ARRAY[1..5] OF LREAL:=[5(10.0)];
	m_instruKiLimit:ARRAY[1..5] OF LREAL:=[5(250.0)];
	m_instruCtrlLimit:ARRAY[1..5] OF LREAL:=[5(400.0)];
	
	// max grip force/current(mA)
	m_maxGripForce:LREAL;
	m_maxGripCurrent:LREAL:=400.0;
	
	// max gripper finger control force/current(mA)
	m_maxGripCtrlForce:LREAL;
	m_maxGripCtrlCurrent:LREAL:=400.0;
	
	// PID for instrument joint position
	m_instruJntCtrl:ARRAY[1..5] OF FB_PID;

	// command instrument joint position and velocity
	m_instruCmdJntPos:Vec5d;
	m_instruLastCmdJntPos:Vec5d;
	m_instruCmdJntVel:Vec5d;
	
	// current instrument joint position and velocity
	m_instruCurJntPos: Vec5d;
	m_instruCurJntVel:Vec5d;
	
	// grasp force level
	m_graspForceLevel:Lreal :=0;
	
	// instrument joint control torque(when gripper is open)
	m_instruJntCtrlTrq:Vec5d:=[5(0.0)];

END_VAR

METHOD init : BOOL
VAR_IN_OUT CONSTANT
	i_slaveArm:FB_SlaveArm;
END_VAR

VAR
	i,j:INT;
	currentRatioMotor2Jnt:LREAL;
END_VAR
m_graspForceLevel:=0;

// init controller
currentRatioMotor2Jnt:=GVL_SlaveMotorParameters.g_motorTrqConst[4]*GVL_SlaveMotorParameters.g_motorReduction[4]/1000;
m_maxGripForce := m_maxGripCurrent * currentRatioMotor2Jnt;
m_maxGripCtrlForce := m_maxGripCtrlCurrent * currentRatioMotor2Jnt;
FOR i:=1 TO 5 DO
	m_instruCmdJntPos[i]:=i_slaveArm.curJntPos[i+3];
	m_instruLastCmdJntPos[i]:=m_instruCmdJntPos[i];
	m_instruCmdJntVel[i]:=0;
	
	m_instruJntCtrl[i].init(g_slaveArmCtrlCycleTime,m_instruKp[i],m_instruKd[i],m_instruKi[i],
		m_instruKiLimit[i]* currentRatioMotor2Jnt,	m_instruCtrlLimit[i]*currentRatioMotor2Jnt);
END_FOR
END_METHOD

METHOD run : BOOL
VAR_IN_OUT CONSTANT
	// instrument joint command position
	i_cmdInstruJntPos :Vec5d;
	
	// instrument joint command velocity
	i_cmdInstruJntVel :Vec5d;
	
	// command grip force level
	i_cmdGripForceLevel:LREAL;
	
	// slave arm data
	i_slaveArm :FB_SlaveArm;
END_VAR

VAR_OUTPUT
	// joint control torque
	o_cmdJntTrq:Vec5d;
END_VAR

VAR
	i: INT;
END_VAR
m_graspForceLevel:=LIMIT(0,i_cmdGripForceLevel ,  100)	;

// joint position control
FOR i:=1 TO 5 DO	
	m_instruCmdJntPos[i]:=i_cmdInstruJntPos[i];
	m_instruCmdJntVel[i]:=i_cmdInstruJntVel[i];
	m_instruCurJntPos[i]:=i_slaveArm.curJntPos[i+3];
	m_instruCurJntVel[i]:= i_slaveArm.curJntVel[i+3];
	m_instruJntCtrlTrq[i]:=m_instruJntCtrl[i].run(m_instruCmdJntPos[i],m_instruCurJntPos[i], m_instruCmdJntVel[i], m_instruCurJntVel[i]);
END_FOR
m_instruJntCtrlTrq[1]:=0;
m_instruJntCtrlTrq[2]:=0;
m_instruJntCtrlTrq[4]:=0;

// exert grip force 
IF m_graspForceLevel >0  THEN
	m_instruJntCtrlTrq[3]:= -m_maxGripForce*m_graspForceLevel/100.0;	
END_IF

o_cmdJntTrq := m_instruJntCtrlTrq;
END_METHOD

END_FUNCTION_BLOCK

// ---- FBs_SlaveControllers/FB_SlaveCtrlInstruCali.TcPOU
// Brief: Calibrate the zero position of Instrument
FUNCTION_BLOCK PUBLIC FB_SlaveCtrlInstruCali EXTENDS FB_SlaveArmCtrlBase
VAR
	// flag to start calibration
	m_instruCaliStart:BOOL;
	
	// mount motion planning
	m_jntOTG :ARRAY[1..8] OF FB_secOrdTrajFilter;
	m_instruMountVel :LREAL := 1*PI;
	m_instruMountAcc :LREAL := 2*PI;

	// 	cali status
	m_rollJntCaliStatus :INT := 0;
	m_pitchJntCaliStatus :INT := 0;
	m_yawJntCaliStatus :INT := 0;
	
	// flag if zero position is written to CoE
	m_zeroPosWritten :BOOL;
	m_zeroPosWriteStart :BOOL;
	
	// flag if SN is written to CoE
	m_SNWritten:BOOL;
	m_SNWriteStart:BOOL;
	
	// joint current threshold which indicate panel is buckled with instrument
	m_maxJntCurrent :LREAL := 300;
	
	// joint current threshold which indicate finger closed
	m_fingerCloseCurrent :LREAL := 50;
	
	// joint position at limits
	m_jntLimitPos1, m_jntLimitPos2, m_jntCaliPos :LREAL;
	m_jntLimitPos3, m_jntLimitPos4 :LREAL;

	// flag if joint is mounted
	m_jointMounted :ARRAY[1..8] OF BOOL := [5(FALSE)];
	
	// instrument mount motion range
	m_mountMotionAng :LREAL :=30*g_deg2Rad;
	
	// command mount motion
	m_targetMountPos :Vec8d;
	
	// instrument zero position
	m_instruZeroPosition :Vec5d;
	
	// angle to close finger
	m_baseCloseAngle :LREAL := 1*g_deg2Rad;
	m_bipolarCloseAngle :LREAL := 5*g_deg2Rad;
	m_proGraspCloseAngle:LREAL := 25*g_deg2Rad;
	
	//new endoscope calibration
	m_scopeMountStatus :INT := 0;
	// instrument zero position
	m_instruZeroDeviation :Vec5d;
	m_maxJntCurrentEndoscope :Vec5d := [120, 120, 120, 120, 120];
	newEndoscopeCaliCompelet: BOOL:=FALSE;
	
	
	m_gripAngleOTG : FB_secOrdTrajFilter;
	m_targetGripAng:LREAL;
	m_cmdGripAng:LREAL;
	m_cmdDHJntPos :Vec6d;
	m_initTrig:R_TRIG;
	m_cmdJntPosMid:Vec8d;
	
	A:LREAL;
END_VAR

// override this function in each exact controller
METHOD PROTECTED calcCmdJntPos : BOOL
VAR_IN_OUT CONSTANT
	i_endoscopePose : ST_Frame;
	i_masterStatus :ST_MasterStatus;
	i_setupStatus: ST_SetupStatus;
	i_slaveArm :FB_SlaveArm;
END_VAR

VAR 
	i :INT;
END_VAR
// retur directly if instrument/endoscope is not readed
IF NOT i_slaveArm.instrument.onChipData.m_InstruReadSucceed THEN
	m_rollJntCaliStatus :=0;
	m_pitchJntCaliStatus :=0;
	m_yawJntCaliStatus :=0;
	m_scopeMountStatus:=0;
	m_zeroPosWritten :=FALSE;
	m_zeroPosWriteStart:=FALSE;
	m_SNWritten :=FALSE;
	m_SNWriteStart:=FALSE;
	m_instruCaliStart:=FALSE;
	m_jntOPMode[6] := DriverOPMode_PosTrq;
	m_jntOPMode[7] := DriverOPMode_PosTrq;
	FOR i:=4 TO 8 DO
		m_jointMounted[i]:=FALSE;
	END_FOR
	return;
END_IF
m_initTrig(CLK:=m_yawJntCaliStatus = -1);
IF m_initTrig.Q THEN
	m_targetGripAng := i_slaveArm.curGripAngle;
	m_gripAngleOTG.init(m_targetGripAng, 0, 2*m_instruMountVel, 10*m_instruMountAcc, g_slaveArmCtrlCycleTime);
END_IF
IF m_yawJntCaliStatus = -1 THEN
	jog(i_slaveArm);
END_IF
// write zero position to CoE
IF GVL_InstruTestUIVars.g_writeZeroPosFlag THEN
	GVL_InstruTestUIVars.g_writeZeroPosFlagErr:=0;
	IF ABS(i_slaveArm.filtJntCurrent[4])<150 AND ABS(i_slaveArm.filtJntCurrent[5])<150 THEN
		m_zeroPosWriteStart := TRUE;
	ELSE
		GVL_InstruTestUIVars.g_writeZeroPosFlagErr:=1;
	END_IF
ELSE
	IF (m_yawJntCaliStatus = -1 OR m_scopeMountStatus = -1) AND m_zeroPosWriteStart THEN
		IF NOT m_zeroPosWritten THEN
			IF InstruType_NewEndoscope = i_slaveArm.instrument.onChipData.m_InstruID THEN
				FOR  i:=1 TO  5 DO
					m_instruZeroPosition[i]:=i_slaveArm.linkSingle[i+3];
				END_FOR
				m_zeroPosWritten := i_slaveArm.instrument.writeZeroPosToChip(m_instruZeroPosition[4],0.0,0.0);
			ELSE
				m_zeroPosWritten := i_slaveArm.instrument.writeZeroPosToChip(m_instruZeroPosition[1],m_instruZeroPosition[2],m_instruZeroPosition[3]);
			END_IF
				
		ELSE
			m_zeroPosWriteStart:=FALSE;
			m_zeroPosWritten:=FALSE;
		END_IF
		RETURN;
	END_IF;
END_IF


// move joint to zero position
IF GVL_InstruTestUIVars.g_searchZeroPosFlag THEN
	m_rollJntCaliStatus :=0;
	m_pitchJntCaliStatus :=0;
	m_yawJntCaliStatus :=0;
	m_instruCaliStart := TRUE;
ELSE
	IF m_instruCaliStart THEN
		// calibrate motion
		IF InstruType_NewEndoscope = i_slaveArm.instrument.onChipData.m_InstruID THEN
			newEndoscopeCali(i_slaveArm);
			IF m_scopeMountStatus = -1 THEN
				m_jntOPMode[6] := DriverOPMode_Trq;
				m_jntOPMode[7] := DriverOPMode_Trq;
				GVL_InstruTestUIVars.g_instruCaliState:=TRUE;
				m_instruZeroPosition[1]:=0;
				m_instruZeroPosition[2]:=0;
				m_instruZeroPosition[3]:=0;
				m_instruZeroPosition[4]:=i_slaveArm.linkSingle[7];
				m_instruZeroPosition[5]:=0;
				GVL_InstruTestUIVars.writeInstruZeroPos:=m_instruZeroPosition;
				m_instruCaliStart:=FALSE;
			END_IF
			
		ELSE
			IF m_rollJntCaliStatus <> -1 THEN
				rollJntCali(i_slaveArm);
			ELSIF m_pitchJntCaliStatus <> -1 THEN
				pitchJntCali(i_slaveArm);
			ELSIF m_yawJntCaliStatus <> -1 THEN
				IF  i_slaveArm.instrument.instruTypeInfo.m_isSingleFinger THEN
					yawJntCali_finger(i_slaveArm);
				ELSE
					yawJntCali_gripper(i_slaveArm);
				END_IF
			
			END_IF
			
			// calibrate motion finish and record position
			IF m_yawJntCaliStatus = -1 THEN
				FOR  i:=1 TO  5 DO
					m_instruZeroPosition[i]:=i_slaveArm.linkSingle[i+3];
				END_FOR
				GVL_InstruTestUIVars.g_instruCaliState:=TRUE;
				GVL_InstruTestUIVars.writeInstruZeroPos:=m_instruZeroPosition;
				m_instruCaliStart:=FALSE;
			END_IF
		END_IF
		
	END_IF
		
END_IF

IF m_yawJntCaliStatus = -1 THEN
	FOR  i:=1 TO  5 DO
		m_instruZeroPosition[i]:=i_slaveArm.linkSingle[i+3];
	END_FOR
	GVL_InstruTestUIVars.writeInstruZeroPos:=m_instruZeroPosition;
END_IF
END_METHOD

PROPERTY getState : BOOL
GET
getState:=m_instruCaliStart;(*(m_yawJntCaliStatus <> -1 AND m_scopeMountStatus <> -1)AND 
		  (m_rollJntCaliStatus<>0 OR m_pitchJntCaliStatus<>0 OR m_yawJntCaliStatus<>0 OR m_scopeMountStatus<>0);*)
END_GET
END_PROPERTY

METHOD PUBLIC init : BOOL
VAR_IN_OUT CONSTANT
	i_slaveArm	:FB_SlaveArm;
END_VAR
VAR_IN_OUT 
	r_slaveArmCtrlCmd :ST_SlaveArmCtrlCmds;
END_VAR

VAR
	i : INT;
END_VAR
// check if to hold the command joint position unchanged
m_holdLastCmds := checkToHoldLastCmds(i_slaveArm);

SUPER^.Init(i_slaveArm,r_slaveArmCtrlCmd);
m_jntOPMode[4] := DriverOPMode_PosTrq;
m_jntOPMode[5] := DriverOPMode_PosTrq;
m_jntOPMode[6] := DriverOPMode_PosTrq;
m_jntOPMode[7] := DriverOPMode_PosTrq;
m_jntOPMode[8] := DriverOPMode_PosTrq;
FOR i:=1 TO 8 DO
	m_targetMountPos[i]:=m_cmdJntPos[i];
	m_jntOTG[i].init(m_targetMountPos[i], 0,m_instruMountVel, m_instruMountAcc, g_slaveArmCtrlCycleTime);
	m_jointMounted[i]:=FALSE;
END_FOR

m_rollJntCaliStatus :=0;
m_pitchJntCaliStatus :=0;
m_yawJntCaliStatus :=0;
m_zeroPosWritten := FALSE;
GVL_InstruTestUIVars.g_writeZeroPosFlagErr:=0;

m_zeroPosWriteStart:=FALSE;
m_SNWritten :=FALSE;
m_SNWriteStart:=FALSE;
m_instruCaliStart:=FALSE;
newEndoscopeCaliCompelet:=FALSE;
m_scopeMountStatus:=0;

IF i_slaveArm.instrument.instruType = InstruType_Endoscope OR i_slaveArm.instrument.instruType = InstruType_NewEndoscope THEN
	m_jntEnableFlag := g_zeroVec8i;
	m_rollJntCaliStatus := -1;
	m_pitchJntCaliStatus := -1;
	m_yawJntCaliStatus := -1;
	m_scopeMountStatus := -1;
ELSE 
	m_jntEnableFlag := g_onesVec8i;
END_IF
m_jntEnableFlag[1] := 0;
m_jntEnableFlag[2] := 0;
m_jntEnableFlag[3] := 0;

// update commands to arm
copyCmds(r_slaveArmCtrlCmd);
END_METHOD

METHOD jog : BOOL
VAR_IN_OUT CONSTANT
	i_slaveArm :FB_SlaveArm;
END_VAR

VAR 

END_VAR
IF GVL_InstruTestUIVars.g_jogClose THEN
//	m_targetGripAng:=i_slaveArm.curGripAngle-1*g_deg2Rad;
	GVL_InstruTestUIVars.g_jogClose:=0;
	IF InstruType_ProGraspForceps = i_slaveArm.instrument.onChipData.m_InstruID THEN
		m_cmdJntPos[4]:=m_cmdJntPos[4]+ASIN((2.8/5.26) * SIN(1*i_slaveArm.instrument.instruTypeInfo.m_k1*g_deg2Rad));
		m_cmdJntPos[5]:=m_cmdJntPos[5]+ASIN((2.8/5.26) * SIN(1*i_slaveArm.instrument.instruTypeInfo.m_k1*g_deg2Rad));
	ELSE
		m_cmdJntPos[4]:=m_cmdJntPos[4]+1*g_deg2rad*i_slaveArm.instrument.instruTypeInfo.m_k1;
		m_cmdJntPos[5]:=m_cmdJntPos[5]+1*g_deg2rad*i_slaveArm.instrument.instruTypeInfo.m_k1;
	END_IF
END_IF

RETURN;

m_cmdDHJntPos:=i_slaveArm.curDHJntPos;
jog:=ABS(m_targetGripAng-m_cmdGripAng)<g_jntCtrlAngTolLow;
// traj plan
m_gripAngleOTG.run(m_targetGripAng,0.0, o_cmdAcc=>,o_cmdVel=>,o_cmdPos=>m_cmdGripAng);

// calculate target motor joint position from DH joint position
i_slaveArm.instrument.instruIK(m_cmdDHJntPos,m_cmdGripAng, o_jntPos=>m_cmdJntPosMid);
m_cmdJntPos[4]:=m_cmdJntPosMid[4];
m_cmdJntPos[5]:=m_cmdJntPosMid[5];
END_METHOD

METHOD newEndoscopeCali : BOOL
VAR_IN_OUT CONSTANT
	i_slaveArm :FB_SlaveArm;
END_VAR

VAR 
	i :INT;
	curJntPos :Vec8d;
END_VAR
curJntPos := i_slaveArm.curJntPos;

CASE m_scopeMountStatus OF
	//fix scope lock joint(joint 7)
	0:
		// other joints stay still
		FOR i:=1 TO 5 DO
			IF i = 1 OR i =2 OR i =5 THEN
				m_jointMounted[i] := TRUE;
				m_targetMountPos[i+3]:=curJntPos[i+3];
				m_jntOTG[i].init(m_targetMountPos[i+3], 0,m_instruMountVel, m_instruMountAcc, g_slaveArmCtrlCycleTime);
			END_IF
		END_FOR
	
		// check if buckled
		m_jointMounted[3]:=FALSE; 
		m_jointMounted[4]:=FALSE; 
		FOR i:=3 TO 4 DO
			IF ABS(i_slaveArm.filtJntCurrent[i+3])> m_maxJntCurrentEndoscope[i] THEN 
				m_jointMounted[i]:=TRUE;
				m_targetMountPos[i+3]:=curJntPos[i+3];
				m_jntOTG[i].init(m_targetMountPos[i+3], 0,m_instruMountVel, m_instruMountAcc, g_slaveArmCtrlCycleTime);
				
			ELSE
				m_targetMountPos[i+3]:=curJntPos[i+3]+m_mountMotionAng;
			END_IF
		END_FOR
		
		IF m_jointMounted[3] AND m_jointMounted[4] THEN
			m_scopeMountStatus:=1;
		END_IF
		

	1: // buckle scope rotate joint (joint 8)
		m_jntOPMode[6] := DriverOPMode_Trq;
		m_instruZeroDeviation[4] :=  i_slaveArm.linkSingle[7] - 5.25;
		m_scopeMountStatus :=2;

	2:// move back to zero position
		
		//joint4
		IF m_instruZeroDeviation[4]>0 AND m_instruZeroDeviation[4] > pi THEN
			m_instruZeroDeviation[4] := m_instruZeroDeviation[4] - 2*pi;
		ELSIF m_instruZeroDeviation[4]<0 AND m_instruZeroDeviation[4] < -pi THEN
			m_instruZeroDeviation[4] := m_instruZeroDeviation[4] + 2*pi;
		END_IF
		
		m_targetMountPos[7]:=curJntPos[7] - m_instruZeroDeviation[4];
		m_scopeMountStatus :=3;
		
		
	3:
		newEndoscopeCali := FALSE;
		IF ABS(m_targetMountPos[7]-curJntPos[7]) <GVL_SlaveControlParameters.g_jntCtrlAngTolHigh THEN
			// record current joint position as offset for instrument
			i_slaveArm.instrument.initInstruJntPos(i_slaveArm.curJntPos);
			newEndoscopeCali := TRUE;
			m_scopeMountStatus:=-1;
		END_IF
		
END_CASE

// traj plan
FOR i:=1 TO 5 DO
	m_jntOTG[i].run(m_targetMountPos[i+3],0.0, o_cmdAcc=>m_cmdJntAcc[3+i],o_cmdVel=>m_cmdJntVel[3+i],o_cmdPos=>m_cmdJntPos[i+3]);
END_FOR
END_METHOD

METHOD pitchJntCali : BOOL
VAR_IN_OUT CONSTANT
	i_slaveArm :FB_SlaveArm;
END_VAR

VAR 
	i :INT;
	curJntPos :Vec8d;
	jntIdx :INT;
END_VAR
jntIdx:=6;
curJntPos := i_slaveArm.curJntPos;

CASE m_pitchJntCaliStatus OF
	// rotate clockwise
	0:
		m_targetMountPos[jntIdx]:=curJntPos[jntIdx]+m_mountMotionAng;
	
		//buckle joint
		IF i_slaveArm.filtJntCurrent[jntIdx]> m_maxJntCurrent THEN 
			m_jntLimitPos1 := curJntPos[jntIdx];
			m_targetMountPos[jntIdx]:=curJntPos[jntIdx];
			m_jntOTG[jntIdx].init(m_targetMountPos[jntIdx], 0,m_instruMountVel, m_instruMountAcc, g_slaveArmCtrlCycleTime);
			m_pitchJntCaliStatus := 1;
		END_IF
		
	// rotate anticlockwise
	1:
		m_targetMountPos[jntIdx]:=curJntPos[jntIdx]-m_mountMotionAng;
	
		//buckle  joint
		IF i_slaveArm.filtJntCurrent[jntIdx]<- m_maxJntCurrent THEN 
			m_jntLimitPos2 := curJntPos[jntIdx];
			m_targetMountPos[jntIdx]:=curJntPos[jntIdx];
			m_jntOTG[jntIdx].init(m_targetMountPos[jntIdx], 0,m_instruMountVel, m_instruMountAcc, g_slaveArmCtrlCycleTime);
			m_pitchJntCaliStatus := 2;
		END_IF
	
	2:// calculate center/calibarted position
		m_targetMountPos[jntIdx] :=  (m_jntLimitPos1 + m_jntLimitPos2)/2+ i_slaveArm.instrument.instruTypeInfo.m_instruPitchBachlash/2.0;
		m_pitchJntCaliStatus := 3;

	3:
		IF ABS(m_targetMountPos[jntIdx]-curJntPos[jntIdx]) <GVL_SlaveControlParameters.g_jntCtrlAngTolHigh  THEN
			m_pitchJntCaliStatus := -1;
		END_IF
		
END_CASE

// traj plan
m_jntOTG[jntIdx].run(m_targetMountPos[jntIdx],0.0, o_cmdAcc=>m_cmdJntAcc[jntIdx],o_cmdVel=>m_cmdJntVel[jntIdx],o_cmdPos=>m_cmdJntPos[jntIdx]);
END_METHOD

METHOD rollJntCali : BOOL
VAR_IN_OUT CONSTANT
	i_slaveArm :FB_SlaveArm;
END_VAR

VAR 
	i :INT;
	curJntPos :Vec8d;
	jntIdx :INT;
END_VAR
jntIdx:=7;
curJntPos := i_slaveArm.curJntPos;

CASE m_rollJntCaliStatus OF
	// rotate clockwise
	0:
		m_targetMountPos[jntIdx]:=curJntPos[jntIdx]+m_mountMotionAng;
	
		//buckle  joint
		IF i_slaveArm.filtJntCurrent[jntIdx]> m_maxJntCurrent AND ABS(i_slaveArm.curJntVel[jntIdx]) < 1*g_deg2rad  THEN 
			m_jntLimitPos1 := curJntPos[jntIdx];
			m_targetMountPos[jntIdx]:=curJntPos[jntIdx];
			m_jntOTG[jntIdx].init(m_targetMountPos[jntIdx], 0,m_instruMountVel, m_instruMountAcc, g_slaveArmCtrlCycleTime);
			m_rollJntCaliStatus := 1;
		END_IF
		
	// rotate anticlockwise
	1:
		m_targetMountPos[jntIdx]:=curJntPos[jntIdx]-m_mountMotionAng;
	
		//buckle  joint
		IF i_slaveArm.filtJntCurrent[jntIdx]<- m_maxJntCurrent AND ABS(i_slaveArm.curJntVel[jntIdx]) < 1*g_deg2rad   THEN 
			m_jntLimitPos2 := curJntPos[jntIdx];
			m_targetMountPos[jntIdx]:=curJntPos[jntIdx];
			m_jntOTG[jntIdx].init(m_targetMountPos[jntIdx], 0,m_instruMountVel, m_instruMountAcc, g_slaveArmCtrlCycleTime);
			m_rollJntCaliStatus := 2;
		END_IF
	
	2:// calculate center/calibarted positio
		m_targetMountPos[jntIdx] :=  (m_jntLimitPos1 + m_jntLimitPos2)/2;
		m_rollJntCaliStatus := 3;

	3:
		IF ABS(m_targetMountPos[jntIdx]-curJntPos[jntIdx]) <GVL_SlaveControlParameters.g_jntCtrlAngTolHigh  THEN
			m_rollJntCaliStatus := -1;
		END_IF
		
END_CASE

// traj plan
m_jntOTG[jntIdx].run(m_targetMountPos[jntIdx],0.0, o_cmdAcc=>m_cmdJntAcc[jntIdx],o_cmdVel=>m_cmdJntVel[jntIdx],o_cmdPos=>m_cmdJntPos[jntIdx]);
END_METHOD

METHOD yawJntCali_finger : BOOL
VAR_IN_OUT CONSTANT
	i_slaveArm :FB_SlaveArm;
END_VAR

VAR 
	i :INT;
	curJntPos :Vec8d;
	jntIdx :INT;
END_VAR
jntIdx:=5;
curJntPos := i_slaveArm.curJntPos;

CASE m_yawJntCaliStatus OF
	// rotate clockwise
	0:
		m_targetMountPos[jntIdx]:=curJntPos[jntIdx]+m_mountMotionAng;
	
		//buckle  joint
		IF i_slaveArm.filtJntCurrent[jntIdx]> m_maxJntCurrent THEN 
			m_jntLimitPos1 := curJntPos[jntIdx];
			m_targetMountPos[jntIdx]:=curJntPos[jntIdx];
			m_jntOTG[jntIdx].init(m_targetMountPos[jntIdx], 0,m_instruMountVel, m_instruMountAcc, g_slaveArmCtrlCycleTime);
			m_yawJntCaliStatus := 1;
		END_IF
		
	// rotate anticlockwise
	1:
		m_targetMountPos[jntIdx]:=curJntPos[jntIdx]-m_mountMotionAng;
	
		//buckle  joint
		IF i_slaveArm.filtJntCurrent[jntIdx]<- m_maxJntCurrent THEN 
			m_jntLimitPos2 := curJntPos[jntIdx];
			m_targetMountPos[jntIdx]:=curJntPos[jntIdx];
			m_jntOTG[jntIdx].init(m_targetMountPos[jntIdx], 0,m_instruMountVel, m_instruMountAcc, g_slaveArmCtrlCycleTime);
			m_yawJntCaliStatus := 2;
		END_IF
	
	2:// calculate center/calibarted positio
		m_targetMountPos[jntIdx] :=  (m_jntLimitPos1 + m_jntLimitPos2)/2+i_slaveArm.instrument.instruTypeInfo.m_instruYawBacklash/2.0;;
		m_yawJntCaliStatus := 3;

	3:
		IF ABS(m_targetMountPos[jntIdx]-curJntPos[jntIdx]) <GVL_SlaveControlParameters.g_jntCtrlAngTolLow  THEN
			m_yawJntCaliStatus := -1;
		END_IF
		
END_CASE

// traj plan
m_jntOTG[jntIdx].run(m_targetMountPos[jntIdx],0.0, o_cmdAcc=>m_cmdJntAcc[jntIdx],o_cmdVel=>m_cmdJntVel[jntIdx],o_cmdPos=>m_cmdJntPos[jntIdx]);
END_METHOD

METHOD yawJntCali_gripper : BOOL
VAR_IN_OUT CONSTANT
	i_slaveArm :FB_SlaveArm;
END_VAR

VAR 
	curJntPos :Vec8d;
	gripCloseAng:LREAL;
END_VAR
curJntPos := i_slaveArm.curJntPos;

// determin finger close angle
IF i_slaveArm.instrument.instruType = InstruType_MarylandForceps OR i_slaveArm.instrument.instruType = InstruType_FenestratedForceps
	OR i_slaveArm.instrument.instruType = InstruType_CurvedBipolarDissector OR i_slaveArm.instrument.instruType = InstruType_MicroBipolarForceps THEN
	gripCloseAng := m_bipolarCloseAngle;
ELSIF i_slaveArm.instrument.instruType = InstruType_ProGraspForceps OR i_slaveArm.instrument.instruType = InstruType_ForceBipolar THEN
	gripCloseAng := m_proGraspCloseAngle;
ELSE
	gripCloseAng := m_baseCloseAngle;
END_IF

CASE m_yawJntCaliStatus OF
	// buckle joint4 and joint5 by moving toward limit
	0:
		//buckle panel with instrument
		// check if buckled 
		IF i_slaveArm.filtJntCurrent[4]<- m_maxJntCurrent THEN 
			m_jointMounted[4]:=TRUE;
			m_targetMountPos[4]:=curJntPos[4];
			m_jntOTG[4].init(m_targetMountPos[4], 0,m_instruMountVel, m_instruMountAcc, g_slaveArmCtrlCycleTime);
		END_IF
		IF i_slaveArm.filtJntCurrent[5]<- m_maxJntCurrent THEN 
			m_jointMounted[5]:=TRUE;
			m_targetMountPos[5]:=curJntPos[5];
			m_jntOTG[5].init(m_targetMountPos[5], 0,m_instruMountVel, m_instruMountAcc, g_slaveArmCtrlCycleTime);
		END_IF
		
		// set target joint position
		IF FALSE = m_jointMounted[4] THEN
			m_targetMountPos[4]:=curJntPos[4]-m_mountMotionAng;
		END_IF
		IF FALSE = m_jointMounted[5] THEN
			m_targetMountPos[5]:=curJntPos[5]-m_mountMotionAng;
		END_IF

		IF m_jointMounted[4] AND m_jointMounted[5] THEN
			m_yawJntCaliStatus := 1;
			m_jointMounted[4]:=FALSE;
			m_jointMounted[5]:=FALSE;
		END_IF
	// close finger
	1:
		//buckle panel with instrument
		// check if buckled 
		IF i_slaveArm.filtJntCurrent[4]> m_maxJntCurrent THEN 
			m_jointMounted[4]:=TRUE;
			m_targetMountPos[4]:=curJntPos[4];
			m_jntOTG[4].init(m_targetMountPos[4], 0,m_instruMountVel, m_instruMountAcc, g_slaveArmCtrlCycleTime);
		END_IF
		IF i_slaveArm.filtJntCurrent[5]> m_maxJntCurrent THEN 
			m_jointMounted[5]:=TRUE;
			m_targetMountPos[5]:=curJntPos[5];
			m_jntOTG[5].init(m_targetMountPos[5], 0,m_instruMountVel, m_instruMountAcc, g_slaveArmCtrlCycleTime);
		END_IF
		
		// set target joint position
		IF FALSE = m_jointMounted[4] THEN
			m_targetMountPos[4]:=curJntPos[4]+m_mountMotionAng;
		END_IF
		IF FALSE = m_jointMounted[5] THEN
			m_targetMountPos[5]:=curJntPos[5]+m_mountMotionAng;
		END_IF

		IF m_jointMounted[4] AND m_jointMounted[5] THEN
			m_yawJntCaliStatus := 2;
			m_jointMounted[4]:=FALSE;
			m_jointMounted[5]:=FALSE;
		END_IF
		
	2:// move joint5 to open gripper
		m_targetMountPos[4] := curJntPos[4]-i_slaveArm.instrument.instruTypeInfo.m_maxGripAngle/4.0;
		m_targetMountPos[5] := curJntPos[5]-i_slaveArm.instrument.instruTypeInfo.m_maxGripAngle/4.0;
		m_yawJntCaliStatus := 3;

	3:
		IF ABS(m_targetMountPos[5]-curJntPos[5]) <GVL_SlaveControlParameters.g_jntCtrlAngTolLow  THEN
			m_yawJntCaliStatus := 4;
		END_IF
			
	// roll clockwise to reach limit
	4:
		IF NOT(m_jointMounted[4]) THEN  
			// set target joint position
			m_targetMountPos[4]:=curJntPos[4]-m_mountMotionAng;
			// check if reach limit 
			IF i_slaveArm.filtJntCurrent[4]< -m_maxJntCurrent THEN 
				m_jointMounted[4]:=TRUE;
				m_jntLimitPos1 := curJntPos[4];
				m_targetMountPos[4]:=curJntPos[4];
				m_jntOTG[4].init(m_targetMountPos[4], 0,m_instruMountVel, m_instruMountAcc, g_slaveArmCtrlCycleTime);
			END_IF
		END_IF
		IF NOT(m_jointMounted[5]) THEN 
			// set target joint position
			m_targetMountPos[5]:=curJntPos[5]+m_mountMotionAng;
			// check if reach limit 
			IF i_slaveArm.filtJntCurrent[5]> m_maxJntCurrent THEN 
				m_jointMounted[5]:=TRUE;
				m_jntLimitPos2 := curJntPos[5];
				m_targetMountPos[5]:=curJntPos[5];
				m_jntOTG[5].init(m_targetMountPos[5], 0,m_instruMountVel, m_instruMountAcc, g_slaveArmCtrlCycleTime);
			END_IF	
		END_IF
		
		// transit
		IF m_jointMounted[4] AND m_jointMounted[5] THEN
			m_yawJntCaliStatus := 5;
			m_jointMounted[4]:=FALSE;
			m_jointMounted[5]:= FALSE;
		END_IF
		
	5:// move joint5 to open gripper
		m_targetMountPos[5] := curJntPos[5]-i_slaveArm.instrument.instruTypeInfo.m_maxGripAngle/2.0;
		m_yawJntCaliStatus := 6;

	6:
		IF ABS(m_targetMountPos[5]-curJntPos[5]) <GVL_SlaveControlParameters.g_jntCtrlAngTolLow  THEN
			m_yawJntCaliStatus := 7;
		END_IF

